# B&R Automation Studio project NewPendant_NG4_11_05_25A (part 16)

```c
					WRST_TML_Param_Set[i].GlbDirection = 1.0;

					WRST_TML_Param_Set[i].MaxAmpl = 0.0;

				break;

			}
		}

		for(i=0 ; i < 1 ; i++){

			switch(i){

				case 0:

					strcpy(Process[PROC_OSC].Name , "OSC");
					strcpy(VectorStateMach[VECT_OSC].Name , "OSC");

					OSC_TML_Param_Set[i].pPrc = &Process[PROC_OSC];
					OSC_TML_Param_Set[i].pVect = &VectorStateMach[VECT_OSC];
					OSC_TML_Param_Set[i].VectStateNum = 1;
					OSC_TML_Param_Set[i].pTML = &TML_MTR_INST[TML_AX_OSC] ;
					OSC_TML_Param_Set[i].Mode = 1; //BPV Mode

					//OSC_TML_Param_Set[i].MaxOscAmpl = 1.0 * 25.4;
					OSC_TML_Param_Set[i].MaxOscAmpl = 0.0;

				break;

			}

		}

		for(i=0 ; i < 1 ; i++){

			switch(i){

				case 0:

					strcpy(Process[PROC_GAS].Name , "GAS");
					GAS_Param_Set[i].pPrc = &Process[PROC_GAS];

					GAS_Param_Set[i].pSensInput     = &Hardware[1].Inp[5];  //FourAxis Head
					GAS_Param_Set[i].pOutput		= &Hardware[1].Outp[4];

				break;

			}

		}

		for(i=0 ; i < 1 ; i++){

			switch(i){

				case 0:

					strcpy(Process[m->pCfg->HeadCfg.INDX.PROC_Indx].Name , "INDX");
					INDEX_Param_Set[i].pPrc = &Process[m->pCfg->HeadCfg.INDX.PROC_Indx];
					//INDEX_Param_Set[i].pPrc = &Process[PROC_INDX];
					INDEX_Param_Set[i].pVect = &VectorStateMach[m->pCfg->HeadCfg.INDX.VECT_A_Indx];
					strcpy(VectorStateMach[m->pCfg->HeadCfg.INDX.VECT_A_Indx].Name , "INDX A");
					strcpy(VectorStateMach[m->pCfg->HeadCfg.INDX.VECT_B_Indx].Name , "INDX B");
					INDEX_Param_Set[i].VectStateNum = 2;
					INDEX_Param_Set[i].Mode = 0;
					INDEX_Param_Set[i].MaxSpeed = 24.0;
					INDEX_Param_Set[i].pCalibPoints		= &m->pCalib->Points[CALIB_TIG_AMPS_CMD];

				break;

			}

		}

		for(i=0 ; i < 1; i++){

			switch(i){

				case 0:

					strcpy(Process[PROC_COOL].Name , "COOLANT");
					COOL_Param_Set[i].pPrc = &Process[PROC_COOL];

					COOL_Param_Set[i].pSensInput     = &Hardware[1].Inp[4];  //FourAxis Head
					COOL_Param_Set[i].pOutput		= &Hardware[1].Outp[6];

				break;

			}

		}

		for(i=0 ; i < 1; i++){

			switch(i){

				case 0:

					strcpy(Process[PROC_HW_PS].Name , "HW PS");
					HW_PS_Param_Set[i].pPrc = &Process[PROC_HW_PS];

					HW_PS_Param_Set[i].pCalibPoints		= &m->pCalib->Points[CALIB_HW_AMPS_CMD];
					HW_PS_Param_Set[i].rawCmdMax 		= 16383.0;
					HW_PS_Param_Set[i].AmpCMD_Max 		= 160.0;

				break;

			}

		}

		for(i=0 ; i < 2; i++){

			switch(i){

				case 0:

					strcpy(Process[PROC_WIRE_FEED].Name ,"WrFeed");
					strcpy(VectorStateMach[VECT_WF].Name ,"WrFeed#1");
					strcpy(VectorStateMach[VECT_WF_1].Name ,"WrFeed#2");

					WIRE_Param_Set[i].pPrc = &Process[PROC_WIRE_FEED];
					WIRE_Param_Set[i].pVect = &VectorStateMach[VECT_WF];
					WIRE_Param_Set[i].VectStateNum = 1; //BPV Mode
					WIRE_Param_Set[i].Mode = 1;
					WIRE_Param_Set[i].MaxSpeedJog = TML_MTR_INST[TML_AX_WF]._cfg.maxVel;

					WIRE_Param_Set[i].pSynchMode = &WFSynchMode;
					WIRE_Param_Set[i].pSynchClock = &SynchClckToWF;

					WIRE_Param_Set[i].pCalibPoints	= &m->pCalib->Points[CALIB_WF_SPEED_CMD];

				break;

				case 1:

					strcpy(Process[PROC_WIRE_PULSE].Name ,"WrPulse");
					strcpy(VectorStateMach[VECT_WP].Name ,"WrPulse#1");
					strcpy(VectorStateMach[VECT_WP_1].Name ,"WrPulse#2");
					WIRE_Param_Set[i].Mode = 1; //BPV Mode

					WIRE_Param_Set[i].pPrc = &Process[PROC_WIRE_PULSE];
					WIRE_Param_Set[i].pVect = &VectorStateMach[VECT_WP];
					WIRE_Param_Set[i].VectStateNum = 1;

					WIRE_Param_Set[i].pSynchMode = &WPSynchMode;
					WIRE_Param_Set[i].pSynchClock = &SynchClckToWP;

					WIRE_Param_Set[i].pCalibPoints	= &m->pCalib->Points[CALIB_WP_SPEED_CMD];

				break;

		}

		}

		for(i=0 ; i < 1; i++){

			switch(i){

				case 0:

					strcpy(Process[PROC_TVL].Name , "TVL");
					strcpy(VectorStateMach[VECT_TVL].Name , "TVL");

					TVL_ROT_Param_Set[i].Mode = 1; //BPV Mode
					TVL_ROT_Param_Set[i].MaxSpeedJog = TML_MTR_INST[TML_AX_TVL]._cfg.maxVel;

					TVL_ROT_Param_Set[i].pPrc = &Process[PROC_TVL];
					TVL_ROT_Param_Set[i].pVect = &VectorStateMach[VECT_TVL];
					TVL_ROT_Param_Set[i].VectStateNum = 1;

					TVL_ROT_Param_Set[i].VectModeForJog = vectSt_Mode_Volt;

					TVL_ROT_Param_Set[i].TotalRescaleFactor = 1.0;
					TVL_ROT_Param_Set[i].pCalibPoints = &m->pCalib->Points[CALIB_TVL_SPEED_CMD];

					TVL_ROT_Param_Set[i].pTrackDia = &curCfg->Param[parTVL_TrackDia].val[0];
					TVL_ROT_Param_Set[i].pVelTolerance = &curCfg->Param[parTVL_SpeedTolerane].val[0];

					// TVL in Torq Mode
					TVL_ROT_Param_Set[i].VectModeForJog = vectSt_Mode_Vel;

					TVL_ROT_Param_Set[i].pEncoder = &AxisCh[TML_AX_TVL].curPos;
					TVL_ROT_Param_Set[i].pHomePos = &OLD_MTR_POS[TVL_ENC_HOME];
					TVL_ROT_Param_Set[i].EncPerTick = m->pCfg->HeadCfg.TVL.EncPerTick;
					TVL_ROT_Param_Set[i].EncDir = m->pCfg->HeadCfg.TVL.Enc_Dir;
					TVL_ROT_Param_Set[i].TicksAtHighVel = 20;

					TVL_ROT_Param_Set[i].pSynchMode = &TVLSynchMode;
					TVL_ROT_Param_Set[i].pSynchClock = &SynchClckToTVL;

			break;

	}

	}

	////////////////////////////////////////////
	/*
	Process[PROC_OSC].Disable = 1;
	Process[PROC_OSC].TestMode = 1;
	VectorStateMach[VECT_OSC].simul = 1;
	TML_MTR_INST[TML_AX_OSC].Disable = 1;
	*/

	Process[PROC_WRST].Disable = 0;
	Process[PROC_WRST].TestMode = 0;
	VectorStateMach[VECT_WRST].simul = 0;
	TML_MTR_INST[TML_AX_WRST].Disable = 0;

	////////////////////////////////////////////////////////////
	/// To jest Tylko do proby
	/*
	VectorStateMach[VECT_AVC].simul = 1;
	VectorStateMach[VECT_OSC].simul = 1;
	VectorStateMach[VECT_TVL].simul = 1;
	VectorStateMach[VECT_INDX_1].simul = 1;
	VectorStateMach[VECT_INDX_2].simul = 1;
	VectorStateMach[VECT_WF_1].simul = 1;
	VectorStateMach[VECT_WF].simul = 1;
	VectorStateMach[VECT_WP_1].simul = 1;
	VectorStateMach[VECT_WP].simul = 1;

	VectorStateMach[VECT_AVC].testMode = 1;
	VectorStateMach[VECT_OSC].testMode = 1;
	VectorStateMach[VECT_TVL].testMode = 1;
	VectorStateMach[VECT_INDX_1].testMode = 1;
	VectorStateMach[VECT_INDX_2].testMode = 1;
	VectorStateMach[VECT_WF_1].testMode = 1;
	VectorStateMach[VECT_WF].testMode = 1;
	VectorStateMach[VECT_WP_1].testMode = 1;
	VectorStateMach[VECT_WP].testMode = 1;

	// To tylko trzeba uncomment gdy jest bez torch ale reszta dziala
	TML_MTR_INST[TML_AX_AVC].Disable = 1;
	TML_MTR_INST[TML_AX_OSC].Disable = 1;
	TML_MTR_INST[TML_AX_TVL].Disable = 1;
	TML_MTR_INST[TML_AX_WRST].Disable = 1;
	TML_MTR_INST[TML_AX_WF].Disable = 1;
	TML_MTR_INST[TML_AX_WF_1].Disable = 1;
	TML_MTR_INST[TML_AX_WP].Disable = 1;
	TML_MTR_INST[TML_AX_WP_1].Disable = 1;
	////////////////////////////////////////

	Process[PROC_AVC].Disable = 1;
	Process[PROC_AVC].TestMode = 1;

	Process[PROC_INDX].Disable = 1;
	Process[PROC_INDX].TestMode = 1;

	Process[PROC_OSC].Disable = 1;
	Process[PROC_OSC].TestMode = 1;

	Process[PROC_TVL].Disable = 1;
	Process[PROC_TVL].TestMode = 1;

	Process[PROC_WIRE_FEED].Disable = 1;
	Process[PROC_WIRE_FEED].TestMode = 1;

	Process[PROC_WIRE_PULSE].Disable = 1;
	Process[PROC_WIRE_PULSE].TestMode = 1;

	Process[PROC_COOL].Disable = 1;
	Process[PROC_COOL].TestMode = 1;

	Process[PROC_GAS].Disable = 1;
	Process[PROC_GAS].TestMode = 1;
	*/
	////////////////////////////////////////////////////////

	return 1;

}

DINT Configure_CLAMSHELL_HEAD(MASTER_typ * m, UINT headType){
int i;

CurCfg_typ *curCfg;
Cfg_typ *cfg;
CurCalib_typ *curCalib , *defaultCalib;

	if(!m)
		return;

	curCfg = (CurCfg_typ*)m->pCurCfg;
	cfg = (Cfg_typ*)m->pCfg;

	curCalib = m->pCalib;
	defaultCalib = m->pDefaultCalib;

	if(!curCfg || !cfg || !curCalib  || !defaultCalib)
		return;

/*********************************************/
	/***   Hardware and Vectors *********************/

	TML_MTR_INST[m->pCfg->HeadCfg.TVL.TML_Indx ].pState = &VectorStateMach[m->pCfg->HeadCfg.TVL.VECT_Indx];

	TML_MTR_INST[m->pCfg->HeadCfg.AVC.TML_A_Indx ].pState = &VectorStateMach[m->pCfg->HeadCfg.AVC.VECT_A_Indx];
	TML_MTR_INST[m->pCfg->HeadCfg.AVC.TML_B_Indx ].pState = &VectorStateMach[m->pCfg->HeadCfg.AVC.VECT_B_Indx];

	TML_MTR_INST[m->pCfg->HeadCfg.OSC.TML_A_Indx ].pState = &VectorStateMach[m->pCfg->HeadCfg.OSC.VECT_A_Indx];
	TML_MTR_INST[m->pCfg->HeadCfg.OSC.TML_B_Indx ].pState = &VectorStateMach[m->pCfg->HeadCfg.OSC.VECT_B_Indx];

	TML_MTR_INST[m->pCfg->HeadCfg.WF.TML_A_Indx ].pState = &VectorStateMach[m->pCfg->HeadCfg.WF.VECT_A_Indx];
	TML_MTR_INST[m->pCfg->HeadCfg.WF.TML_B_Indx ].pState = &VectorStateMach[m->pCfg->HeadCfg.WF.VECT_B_Indx];

	TML_MTR_INST[m->pCfg->HeadCfg.WP.TML_A_Indx ].pState = &VectorStateMach[m->pCfg->HeadCfg.WP.VECT_A_Indx];
	TML_MTR_INST[m->pCfg->HeadCfg.WP.TML_B_Indx ].pState = &VectorStateMach[m->pCfg->HeadCfg.WP.VECT_B_Indx];

	TML_MTR_INST[m->pCfg->HeadCfg.WRST.TML_A_Indx ].pState = &VectorStateMach[m->pCfg->HeadCfg.WRST.VECT_A_Indx];
	TML_MTR_INST[m->pCfg->HeadCfg.WRST.TML_B_Indx ].pState = &VectorStateMach[m->pCfg->HeadCfg.WRST.VECT_B_Indx];

	DC_Mtr[m->pCfg->HeadCfg.INDX.DC_A_Indx ].pState = &VectorStateMach[m->pCfg->HeadCfg.INDX.VECT_A_Indx];
	DC_Mtr[m->pCfg->HeadCfg.INDX.DC_B_Indx ].pState = &VectorStateMach[m->pCfg->HeadCfg.INDX.VECT_B_Indx];

	/*********************************************************/
	/****   Phisical hardware configuration   ************************/

		for(i = 0 ; i < PROCESS_NUM; i++)
			strcpy(Process[i].Name , "spare");

		for(i = 0 ; i < VECTORS_NUM; i++)
			strcpy(VectorStateMach[i].Name , "spare");

			/***********************************/

		//////////////////////////////////////////////////////////////////////////////////
		// Wire Block
		for(i=0 ; i < 2; i++){

			switch(i){

				case 0:
					strcpy(Process[m->pCfg->HeadCfg.WB[i].PROC_Indx].Name , "WB_UD");
					strcpy(VectorStateMach[m->pCfg->HeadCfg.WB[i].VECT_Indx].Name , "WB_UD");

					WR_BLK_Param_Set[i].pPrc = &Process[m->pCfg->HeadCfg.WB[i].PROC_Indx];
					WR_BLK_Param_Set[i].pVect = &VectorStateMach[m->pCfg->HeadCfg.WB[i].VECT_Indx];
					WR_BLK_Param_Set[i].VectStateNum = 1;

					WR_BLK_Param_Set[i].MaxSpeedJog = 24.0;

					Gen_one = 1.0;
					WR_BLK_Param_Set[i].pJogSpeed = &Gen_one;

				break;

				case 1:
					strcpy(Process[m->pCfg->HeadCfg.WB[i].PROC_Indx].Name , "WB_LR");
					strcpy(VectorStateMach[m->pCfg->HeadCfg.WB[i].VECT_Indx].Name , "WB_LR");

					WR_BLK_Param_Set[i].pPrc = &Process[PROC_WB_LR];
					WR_BLK_Param_Set[i].pVect = &VectorStateMach[VECT_WB_LR];
					WR_BLK_Param_Set[i].VectStateNum = 1;

					WR_BLK_Param_Set[i].MaxSpeedJog = 24.0;

					Gen_one = 1.0;
					WR_BLK_Param_Set[i].pJogSpeed = &Gen_one;

				break;

			}

		}

		for(i = 0 ; i < DC2DIRMTR_NUM; i++){

			switch(i){

				case DC_WB_UD:

					strcpy(DC2DirMtr[i].Name , "WB_UD");
					DC2DirMtr[i].pState = &VectorStateMach[VECT_WB_UD];

					DC2DirMtr[i].Cfg.pQ1_output = &Hardware[1].Outp[12];
					DC2DirMtr[i].Cfg.pQ2_output = &Hardware[1].Outp[13];
					DC2DirMtr[i].Cfg.pQ3_output = &Hardware[1].Outp[14];
					DC2DirMtr[i].Cfg.pQ4_output = &Hardware[1].Outp[15];

					DC2DirMtr[i].Cfg.MtrDir = 1.0;

				break;

				case DC_WB_LR:

					strcpy(DC2DirMtr[i].Name , "WB_LR");
					DC2DirMtr[i].pState = &VectorStateMach[VECT_WB_LR];

					DC2DirMtr[i].Cfg.pQ1_output = &Hardware[1].Outp[16];
					DC2DirMtr[i].Cfg.pQ2_output = &Hardware[1].Outp[17];
					DC2DirMtr[i].Cfg.pQ3_output = &Hardware[1].Outp[18];
					DC2DirMtr[i].Cfg.pQ4_output = &Hardware[1].Outp[19];

					DC2DirMtr[i].Cfg.MtrDir = 1.0;

				break;

			}

		}
		/////////////////////////////////////////////////////////////////////////////////

		for(i = 0 ; i < GEN_MTR_NUM; i++){

			switch(i){

				case DC_INDX_1:
				case DC_INDX_2:

					switch(i){

						case DC_INDX_1:

							strcpy(DC_Mtr[i].Name , "DC INDX #1");

							DC_Mtr[i].Cfg.mtr_dir = 1.0;

							if(ProjectConfig == project_US_Orbital) // US Orbital has B and /B swapped
								DC_Mtr[i].Cfg.enc_dir = 1.0;
							else
								DC_Mtr[i].Cfg.enc_dir = -1.0;

							//DC_Mtr[i].Cfg.enc_dir = -1.0;

						break;

						case DC_INDX_2:

							strcpy(DC_Mtr[i].Name , "DC INDX #2");

							DC_Mtr[i].Cfg.mtr_dir = -1.0;

							if(ProjectConfig == project_US_Orbital) // US Orbital has B and /B swapped
								DC_Mtr[i].Cfg.enc_dir = -1.0;
							else
								DC_Mtr[i].Cfg.enc_dir = 1.0;

							//DC_Mtr[i].Cfg.enc_dir = 1.0;

						break;

					}

					//DC_Mtr[i].Cfg.units = 2000 / 59.847340050885561192713356451475; // 2000 enc ticks / 0.75 " dia * 25.4 * PI
					//DC_Mtr[i].Cfg.rev_scale = 66.0 * 0.218686666; // Ratio gear box 66:1

					DC_Mtr[i].Cfg.units =48000 / (1.25 * M_PI * 25.4); // 48000 enc ticks / 1.25 " dia * 25.4 * PI
					DC_Mtr[i].Cfg.rev_scale = 1; // Ratio gear box 66:1

					/* Parameters for PID controller */
					// To nowe
					DC_Mtr[i].msc.PIDParameters.Kp= 100.0;//0.4; //proportional gain / was 0.6
					DC_Mtr[i].msc.PIDParameters.Tn= 0.0;//0.3.1; //intergral action time
					DC_Mtr[i].msc.PIDParameters.Kfbk = 0.1; //windup dampenin

					DC_Mtr[i].msc.PID.enable = 0;
					DC_Mtr[i].msc.PID.pPar = &DC_Mtr[i].msc.PIDParameters;
					DC_Mtr[i].msc.PID.request = 3; // Read parameters from PIDParameters
					DC_Mtr[i].msc.PIDParameters.Tv= 0; //derivative action time
					DC_Mtr[i].msc.PIDParameters.Y_max = 100.0;	//max manipulated variable %
					DC_Mtr[i].msc.PIDParameters.Y_min = -100.0; //min manipulated variable %

				break;

				default:

					strcpy(DC_Mtr[i].Name , "Spare ");

				break;

			}

				//CalcUnits(&DC_Mtr[i]);
				DC_Mtr[i].msc.kPos = (float)DC_Mtr[i].Cfg.units * DC_Mtr[i].Cfg.rev_scale;

		}

		for(i = 0 ; i < TML_SERVO_NUM ; i++){

			switch(i){

				case TML_AX_TVL:

					strcpy(TML_MTR_INST[i].Name , "TVL");

					TML_MTR_INST[i]._cfg.loopPeriod = 0.0005; // Slow loop
					TML_MTR_INST[i]._cfg.units = 1024 * 4; //
					TML_MTR_INST[i]._cfg.rev_motor = 546 * 2; // because loopPeriod is 0.0005
					TML_MTR_INST[i]._cfg.rev_scale = 1.0 /( 2.3 * 25.4 * M_PI) ;

					TML_MTR_INST[i]._cfg.maxVel =  4500.0/60.0/TML_MTR_INST[i]._cfg.rev_motor/ TML_MTR_INST[i]._cfg.rev_scale;
					TML_MTR_INST[i]._cfg.maxAcc = TML_MTR_INST[i]._cfg.maxVel * 10.0 ;
					TML_MTR_INST[i]._cfg.absLastPos = OLD_MTR_POS[TVL_LAST_POS];
					TML_MTR_INST[i]._cfg.absFbk = 2;

					TML_MTR_INST[i]._cfg.HeartBeat = 0.08;

					strcpy(TML_MTR_INST[i]._cfg.programName , "3301_CLMSH_TVL.sw");
					TML_MTR_INST[i].ProgramVersion = ASC2UDINT("3301");

					TML_MTR_INST[i].FirmwareVersion = ASC2UDINT("6A2B");  //0x674B
					TML_MTR_INST[i]._cfg.Appl_ID_adr = 0x7FCF;
					TML_MTR_INST[i]._cfg.NotAutoDownload = 1;

				break;

				case TML_AX_OSC:

					strcpy(TML_MTR_INST[i].Name , "OSC");

					// Analog Feedback from REF
					TML_MTR_INST[i]._cfg.loopPeriod = 0.001;

					TML_MTR_INST[i]._cfg.units = 1024 * 4;
					//TML_MTR_INST[i]._cfg.rev_motor = (-75.0/19.0) * 50.0;
					//TML_MTR_INST[i]._cfg.rev_scale = -1.0/ (0.625 * 25.4 *M_PI) ;
					TML_MTR_INST[i]._cfg.rev_motor = -62;
					TML_MTR_INST[i]._cfg.rev_scale = -1.0/ (0.5 * 25.4) ;

					TML_MTR_INST[i]._cfg.maxVel = 8000.0/60.0/TML_MTR_INST[i]._cfg.rev_motor/ TML_MTR_INST[i]._cfg.rev_scale;
					TML_MTR_INST[i]._cfg.maxAcc = TML_MTR_INST[i]._cfg.maxVel * 10.0 ;
					TML_MTR_INST[i]._cfg.absLastPos = OLD_MTR_POS[OSC_LAST_POS];
					TML_MTR_INST[i]._cfg.absFbk = 2;

					TML_MTR_INST[i]._cfg.HeartBeat = 0.4;
					TML_MTR_INST[i]._cfg.PVTPeriod = 0.08;

					strcpy(TML_MTR_INST[i]._cfg.programName , "3302_CLMSH_OSC.sw");
					TML_MTR_INST[i].ProgramVersion = ASC2UDINT("3302");

					TML_MTR_INST[i].FirmwareVersion = ASC2UDINT("6A2B");
					TML_MTR_INST[i]._cfg.Appl_ID_adr = 0x7FCF;
					TML_MTR_INST[i]._cfg.NotAutoDownload = 1;

					//TML_MTR_INST[i]._cfg.sftLimitPos = curCalib->Points[CALIB_OSC_SFT_LIMIT].val[0];
					//TML_MTR_INST[i]._cfg.sftLimitNeg = curCalib->Points[CALIB_OSC_SFT_LIMIT].val[1];

					//TML_MTR_INST[i]._cfg.sftLimitPos = 0.0;
					//TML_MTR_INST[i]._cfg.sftLimitNeg = 0.0;

				break;

				case TML_AX_AVC:
				case TML_AX_AVC2:

					if(i == TML_AX_AVC)
						strcpy(TML_MTR_INST[i].Name , "AVC");
					else
						strcpy(TML_MTR_INST[i].Name , "AVC_2");

					// Analog Feedback from REF
					TML_MTR_INST[i]._cfg.loopPeriod = 0.001;
					TML_MTR_INST[i]._cfg.units = 4096;
					TML_MTR_INST[i]._cfg.rev_motor = 1;
					TML_MTR_INST[i]._cfg.rev_scale = 1.0/5.0;
					TML_MTR_INST[i]._cfg.maxVel = 1500.0;
					TML_MTR_INST[i]._cfg.maxAcc = TML_MTR_INST[i]._cfg.maxVel * 10.0;
					//TML_MTR_INST[i]._cfg.satpMax = 27853; // KPP bylo Stauration of proportional gain
					TML_MTR_INST[i]._cfg.satpMax = 32000; // KPP bylo Stauration of proportional gain
					//TML_MTR_INST[i]._cfg.kppMax = 32000; // KPP bylo Stauration of proportional gain
					//TML_MTR_INST[i]._cfg.kipMax = 200; // KPP bylo Stauration of proportional gain
					TML_MTR_INST[i]._cfg.kppMax = 32000;
					TML_MTR_INST[i]._cfg.kipMax = 1000;
					TML_MTR_INST[i]._cfg.absFbk = 0;

					TML_MTR_INST[i]._cfg.HeartBeat = 0.8;

					TML_MTR_INST[i]._cfg.signFilter = curCfg->Param[parAVC_FbkFilter].val[0];

					//U_BEND_HP_PINS
					strcpy(TML_MTR_INST[i]._cfg.programName , "3303_CLMSH_AVC.sw");
					TML_MTR_INST[i].ProgramVersion = ASC2UDINT("3303");

					TML_MTR_INST[i].FirmwareVersion = ASC2UDINT("6A2B");  //0x674C , 514D
					TML_MTR_INST[i]._cfg.Appl_ID_adr = 0x7FCF;
					TML_MTR_INST[i]._cfg.NotAutoDownload = 1;

					//TML_MTR_INST[i]._cfg.sftLimitPos = 0.0;
					//TML_MTR_INST[i]._cfg.sftLimitNeg = 0.0;

					/*
					TML_MTR_INST[i]._cfg.AnalLimitPos = 3900;
					TML_MTR_INST[i]._cfg.AnalLimitNeg = 100;
					*/

					TML_MTR_INST[i]._cfg.AnalLimitPos = 0;
					TML_MTR_INST[i]._cfg.AnalLimitNeg = 0;

				break;

				// WRIST
				case TML_AX_WF_1: //TML_AX_WRST:

					strcpy(TML_MTR_INST[i].Name , "WRIST");

					// Analog Feedback from REF
					TML_MTR_INST[i]._cfg.loopPeriod = 0.001;

					TML_MTR_INST[i]._cfg.units = 1024 * 4;
					//TML_MTR_INST[i]._cfg.rev_motor = (-75.0/19.0) * 50.0;
					//TML_MTR_INST[i]._cfg.rev_scale = -1.0/ (0.625 * 25.4 *M_PI) ;
					TML_MTR_INST[i]._cfg.rev_motor = 16 * 50;
					TML_MTR_INST[i]._cfg.rev_scale = 1.0/ (360.0) ;

					TML_MTR_INST[i]._cfg.maxVel = 8000.0/60.0/TML_MTR_INST[i]._cfg.rev_motor/ TML_MTR_INST[i]._cfg.rev_scale;
					TML_MTR_INST[i]._cfg.maxAcc = TML_MTR_INST[i]._cfg.maxVel * 10.0 ;
					TML_MTR_INST[i]._cfg.absLastPos = OLD_MTR_POS[WRST_LAST_POS];
					TML_MTR_INST[i]._cfg.absFbk = 0;
					//TML_MTR_INST[i]._cfg.absFbk = 2;

					TML_MTR_INST[i]._cfg.HeartBeat = 0.02;
					TML_MTR_INST[i]._cfg.PVTPeriod = 0.08;

					strcpy(TML_MTR_INST[i]._cfg.programName , "3307_CLMSH_WRST.sw");
					TML_MTR_INST[i].ProgramVersion = ASC2UDINT("3307");

					TML_MTR_INST[i].FirmwareVersion = ASC2UDINT("6A2B");
					TML_MTR_INST[i]._cfg.Appl_ID_adr = 0x7FCF;
					TML_MTR_INST[i]._cfg.NotAutoDownload = 1;

					//TML_MTR_INST[i]._cfg.sftLimitPos = curCalib->Points[CALIB_OSC_SFT_LIMIT].val[0];
					//TML_MTR_INST[i]._cfg.sftLimitNeg = curCalib->Points[CALIB_OSC_SFT_LIMIT].val[1];

					//TML_MTR_INST[i]._cfg.sftLimitPos = 0.0;
					//TML_MTR_INST[i]._cfg.sftLimitNeg = 0.0;

				break;

				case TML_AX_WF:

					strcpy(TML_MTR_INST[i].Name , "WF");
					TML_MTR_INST[i]._cfg.rev_scale = 1.0 /( 0.75 * 25.4 * M_PI) ;
					TML_MTR_INST[i]._cfg.rev_motor = 35.0;	// jest 39:1 ale trzeba pamietac o groove na rolce

					// Analog Feedback from REF
					TML_MTR_INST[i]._cfg.loopPeriod = 0.001;
					TML_MTR_INST[i]._cfg.units = 1024 * 4; //
					//TML_MTR_INST[i]._cfg.rev_motor = 35;

					TML_MTR_INST[i]._cfg.maxVel = 520 * 25.4/ 60.0; //// 520 ipm
					//TML_MTR_INST[i]._cfg.maxAcc = TML_MTR_INST[i]._cfg.maxVel * 100.0;
					TML_MTR_INST[i]._cfg.maxAcc = TML_MTR_INST[i]._cfg.maxVel * 4.0;
					TML_MTR_INST[i]._cfg.absFbk = 0;

					TML_MTR_INST[i]._cfg.HeartBeat = 0.4;

					strcpy(TML_MTR_INST[i]._cfg.programName , "3305_CLMSH_WF.sw");
					TML_MTR_INST[i].ProgramVersion = ASC2UDINT("3305");

					TML_MTR_INST[i].FirmwareVersion = ASC2UDINT("6A2B");
					TML_MTR_INST[i]._cfg.Appl_ID_adr = 0x7FCF;
					TML_MTR_INST[i]._cfg.NotAutoDownload = 1;

				break;

				case TML_AX_WP:

					strcpy(TML_MTR_INST[i].Name , "WP");

					// Analog Feedback from REF
					TML_MTR_INST[i]._cfg.loopPeriod = 0.001;

					TML_MTR_INST[i]._cfg.units = 1024 * 4;
					TML_MTR_INST[i]._cfg.rev_motor = 3.9;
					TML_MTR_INST[i]._cfg.rev_scale = 1.0/2.0;

					/*
					TML_MTR_INST[i]._cfg.units = 500 * 4;
					TML_MTR_INST[i]._cfg.rev_motor = 24;
					TML_MTR_INST[i]._cfg.rev_scale = 1.0/5.0;
					*/

					TML_MTR_INST[i]._cfg.maxVel = 10000.0; //
					TML_MTR_INST[i]._cfg.maxAcc = 100.0;
					TML_MTR_INST[i]._cfg.absFbk = 0;

					TML_MTR_INST[i]._cfg.HeartBeat = 0.4;

					strcpy(TML_MTR_INST[i]._cfg.programName , "3306_CLMSH_WP.sw");
					TML_MTR_INST[i].ProgramVersion = ASC2UDINT("3306");

					TML_MTR_INST[i].FirmwareVersion = ASC2UDINT("6A2B");
					TML_MTR_INST[i]._cfg.Appl_ID_adr = 0x7FCF;
					TML_MTR_INST[i]._cfg.NotAutoDownload = 1;

				break;

				default:

					//strcpy(TML_MTR_INST[i].Name , "Spare ");
					xsprintf(TML_MTR_INST[i].Name, "Spare %d", i );

				break;

			}

		TML_MTR_INST[i].xCMD = TML_RESTART;

	}

		TML_mgr[0].hrdw[0].AxisNum = 0;
		TML_mgr[0].hrdw[1].AxisNum = 7;

		TML_mgr[0].pAxis[0] = &AxisCh[TML_mgr[0].hrdw[0].AxisNum];
		TML_mgr[0].pAxis[1] = &AxisCh[TML_mgr[0].hrdw[0].AxisNum];
		//TML_mgr[0].pAxis[1] = &AxisCh[TML_mgr[0].hrdw[1].AxisNum];

		TML_mgr[0].pTML[0] = &TML_MTR_INST[0];
		TML_mgr[0].pTML[1] = &TML_MTR_INST[TML_mgr[0].hrdw[0].AxisNum];

		AxisCh[TML_AX_TVL].AxisID	= 1;
		AxisCh[TML_AX_OSC].AxisID 	= 2;
		AxisCh[TML_AX_AVC].AxisID 	= 3;
		AxisCh[TML_AX_AVC2].AxisID 	= 4;

		AxisCh[TML_AX_WF].AxisID 	= 5;
		AxisCh[TML_AX_WP].AxisID 	= 6;

		AxisCh[m->pCfg->HeadCfg.WRST.TML_A_Indx].AxisID 	= 7;

		//AxisCh[TML_AX_WF_1].AxisID 	= 7;
		//AxisCh[TML_AX_WP_1].AxisID 	= 8;
		/**************************************/
		/****   Process   ************************/

		// Lincoln Power Supply
		for(i=0 ; i < 1; i++){

			switch(i){

				case 0:

					strcpy(Process[PROC_TIG_PS].Name , "TIG PS");
					PS_Param_Set[i].pPrc = &Process[PROC_TIG_PS];

					PS_Param_Set[i].pCalibPoints		= &m->pCalib->Points[CALIB_TIG_AMPS_CMD];
					//PS_Param_Set[i].rawCmdMax			= 26170; // //
					//PS_Param_Set[i].AmpCMD_Max			= 500.0; // 62.5 amp / 1 V
					PS_Param_Set[i].rawCmdMax			= 32767;
					PS_Param_Set[i].AmpCMD_Max			= 627.0;

					PS_Param_Set[i].pArcLinkRobot   = (UDINT)&ArcLink.robot;

					PS_Param_Set[i].Mode 			= 1; // Arclink connection

				break;

			}

		}
		///////////////////////////////////////////////////////

		for(i=0 ; i < 1 ; i++){

			switch(i){

				case 0:

					strcpy(Process[PROC_AVC].Name , "AVC");

					strcpy(VectorStateMach[VECT_AVC].Name , "AVC");
					strcpy(VectorStateMach[VECT_AVC2].Name , "AVC_2");

					AVC_Param_Set[i].pPrc = &Process[PROC_AVC];
					AVC_Param_Set[i].pVect = &VectorStateMach[VECT_AVC];
					AVC_Param_Set[i].VectStateNum = 2;
					AVC_Param_Set[i].Mode = 1; //BPV Mode
					AVC_Param_Set[i].Mode = 3; //BPV Mode w/ twp torches
					AVC_Param_Set[i].MaxSpeedJog = TML_MTR_INST[TML_AX_AVC]._cfg.maxVel;

					m->pCalib->Points[CALIB_TIG_VOLT_FBK].num = 10;
					AVC_Param_Set[i].pCalibPoints		= &m->pCalib->Points[CALIB_TIG_VOLT_FBK];

				break;

			}
		}

		for(i=0 ; i < 1 ; i++){

			switch(i){

				case 0:

					strcpy(Process[m->pCfg->HeadCfg.WRST.PROC_Indx].Name , "WRST");
					strcpy(VectorStateMach[m->pCfg->HeadCfg.WRST.VECT_A_Indx].Name , "WRST");

					WRST_TML_Param_Set[i].pPrc = &Process[m->pCfg->HeadCfg.WRST.PROC_Indx];
					WRST_TML_Param_Set[i].pVect = &VectorStateMach[m->pCfg->HeadCfg.WRST.VECT_A_Indx];
					WRST_TML_Param_Set[i].VectStateNum = 1;
					WRST_TML_Param_Set[i].pTML = &TML_MTR_INST[m->pCfg->HeadCfg.WRST.TML_A_Indx] ;
					WRST_TML_Param_Set[i].Mode = 10; // ClamShell Head  mode with Wrist

					WRST_TML_Param_Set[i].GlbDirection = 1.0;

					WRST_TML_Param_Set[i].MaxAmpl = 0.0;

				break;

			}
		}

		for(i=0 ; i < 1 ; i++){

			switch(i){

				case 0:

					strcpy(Process[PROC_OSC].Name , "OSC");
					strcpy(VectorStateMach[VECT_OSC].Name , "OSC");

					OSC_TML_Param_Set[i].pPrc = &Process[PROC_OSC];
					OSC_TML_Param_Set[i].pVect = &VectorStateMach[VECT_OSC];
					OSC_TML_Param_Set[i].VectStateNum = 1;
					OSC_TML_Param_Set[i].pTML = &TML_MTR_INST[TML_AX_OSC] ;
					OSC_TML_Param_Set[i].Mode = 1; //BPV Mode

					//OSC_TML_Param_Set[i].MaxOscAmpl = 1.0 * 25.4;
					OSC_TML_Param_Set[i].MaxOscAmpl = 0.0;

				break;

			}

		}

		for(i=0 ; i < 1 ; i++){

			switch(i){

				case 0:

					strcpy(Process[PROC_GAS].Name , "GAS");
					GAS_Param_Set[i].pPrc = &Process[PROC_GAS];

					//GAS_Param_Set[i].pSensInput     = &Hardware[1].Inp[5];  //FourAxis Head
					//GAS_Param_Set[i].pOutput		= &Hardware[1].Outp[4];

					GAS_Param_Set[i].Mode = 1;// Arclik Gas Sol

				break;

			}

		}

		for(i=0 ; i < 1 ; i++){

			switch(i){

				case 0:

					strcpy(Process[m->pCfg->HeadCfg.INDX.PROC_Indx].Name , "INDX");
					INDEX_Param_Set[i].pPrc = &Process[m->pCfg->HeadCfg.INDX.PROC_Indx];
					//INDEX_Param_Set[i].pPrc = &Process[PROC_INDX];
					INDEX_Param_Set[i].pVect = &VectorStateMach[m->pCfg->HeadCfg.INDX.VECT_A_Indx];
					strcpy(VectorStateMach[m->pCfg->HeadCfg.INDX.VECT_A_Indx].Name , "INDX A");
					strcpy(VectorStateMach[m->pCfg->HeadCfg.INDX.VECT_B_Indx].Name , "INDX B");
					INDEX_Param_Set[i].VectStateNum = 2;
					INDEX_Param_Set[i].Mode = 0;
					INDEX_Param_Set[i].MaxSpeed = 24.0;
					INDEX_Param_Set[i].pCalibPoints		= &m->pCalib->Points[CALIB_TIG_AMPS_CMD];

				break;

			}

		}

		for(i=0 ; i < 1; i++){

			switch(i){

				case 0:

					strcpy(Process[PROC_COOL].Name , "COOLANT");
					COOL_Param_Set[i].pPrc = &Process[PROC_COOL];

					//COOL_Param_Set[i].pSensInput     = &Hardware[1].Inp[4];  //FourAxis Head
					//COOL_Param_Set[i].pOutput		= &Hardware[1].Outp[6];

				break;

			}

		}

		for(i=0 ; i < 1; i++){

			switch(i){

				case 0:

					strcpy(Process[PROC_HW_PS].Name , "HW PS");
					HW_PS_Param_Set[i].pPrc = &Process[PROC_HW_PS];

					HW_PS_Param_Set[i].pCalibPoints		= &m->pCalib->Points[CALIB_HW_AMPS_CMD];

					// small Jack PS
					HW_PS_Param_Set[i].rawCmdMax 		= 16383.0;
					HW_PS_Param_Set[i].AmpCMD_Max 		= 160.0;

					// Lincoln PS
					//HW_PS_Param_Set[i].rawCmdMax 		= 32767.0;
					//HW_PS_Param_Set[i].AmpCMD_Max 		= 160.0;

					HW_PS_Param_Set[i].pAnal_Output 	= &Hardware[1].Anal_Outp[0]; // HotwirePS_AO
					HW_PS_Param_Set[i].pOutput			= &Hardware[1].Outp[2]; //HotwirePS_Enable

				break;

			}

		}

		for(i=0 ; i < 2; i++){

			switch(i){

				case 0:

					strcpy(Process[PROC_WIRE_FEED].Name ,"WrFeed");
					strcpy(VectorStateMach[VECT_WF].Name ,"WrFeed#1");
					strcpy(VectorStateMach[VECT_WF_1].Name ,"WrFeed#2");

					WIRE_Param_Set[i].pPrc = &Process[PROC_WIRE_FEED];
					WIRE_Param_Set[i].pVect = &VectorStateMach[VECT_WF];
					WIRE_Param_Set[i].VectStateNum = 1;
					WIRE_Param_Set[i].Mode = 3; //BPV Mode with Feedback Selection
					WIRE_Param_Set[i].MaxSpeedJog = TML_MTR_INST[TML_AX_WF]._cfg.maxVel;

					WIRE_Param_Set[i].pSynchMode = &WFSynchMode;
					WIRE_Param_Set[i].pSynchClock = &SynchClckToWF;

					WIRE_Param_Set[i].pCalibPoints	= &m->pCalib->Points[CALIB_WF_SPEED_CMD];

				break;

				case 1:

					strcpy(Process[PROC_WIRE_PULSE].Name ,"WrPulse");
					strcpy(VectorStateMach[VECT_WP].Name ,"WrPulse#1");
					strcpy(VectorStateMach[VECT_WP_1].Name ,"WrPulse#2");
					WIRE_Param_Set[i].Mode = 3; //BPV Mode with Feedback Selection

					WIRE_Param_Set[i].pPrc = &Process[PROC_WIRE_PULSE];
					WIRE_Param_Set[i].pVect = &VectorStateMach[VECT_WP];
					WIRE_Param_Set[i].VectStateNum = 1;

					WIRE_Param_Set[i].pSynchMode = &WPSynchMode;
					WIRE_Param_Set[i].pSynchClock = &SynchClckToWP;

					WIRE_Param_Set[i].pCalibPoints	= &m->pCalib->Points[CALIB_WP_SPEED_CMD];

				break;

		}

	}

		for(i=0 ; i < 1; i++){

			switch(i){

				case 0:

					strcpy(Process[PROC_TVL].Name , "TVL");
					strcpy(VectorStateMach[VECT_TVL].Name , "TVL");

					//TVL_ROT_Param_Set[i].Mode = 1; //BPV Mode
					TVL_ROT_Param_Set[i].Mode = 2;  //TVL_MODE_BPV_PosMode
					TVL_ROT_Param_Set[i].MaxSpeedJog = TML_MTR_INST[TML_AX_TVL]._cfg.maxVel;

					TVL_ROT_Param_Set[i].pPrc = &Process[PROC_TVL];
					TVL_ROT_Param_Set[i].pVect = &VectorStateMach[VECT_TVL];
					TVL_ROT_Param_Set[i].VectStateNum = 1;

					TVL_ROT_Param_Set[i].VectModeForJog = vectSt_Mode_Volt;

					TVL_ROT_Param_Set[i].TotalRescaleFactor = 1.0;
					TVL_ROT_Param_Set[i].pCalibPoints = &m->pCalib->Points[CALIB_TVL_SPEED_CMD];

					TVL_ROT_Param_Set[i].pTrackDia = &curCfg->Param[parTVL_TrackDia].val[0];
					TVL_ROT_Param_Set[i].pVelTolerance = &curCfg->Param[parTVL_SpeedTolerane].val[0];

					// TVL in Torq Mode
					TVL_ROT_Param_Set[i].VectModeForJog = vectSt_Mode_Vel;

					TVL_ROT_Param_Set[i].pEncoder = &AxisCh[TML_AX_TVL].curPos;
					TVL_ROT_Param_Set[i].pHomePos = &OLD_MTR_POS[TVL_ENC_HOME];
					TVL_ROT_Param_Set[i].EncPerTick = m->pCfg->HeadCfg.TVL.EncPerTick;
					TVL_ROT_Param_Set[i].EncDir = m->pCfg->HeadCfg.TVL.Enc_Dir;
					TVL_ROT_Param_Set[i].TicksAtHighVel = 20;

					TVL_ROT_Param_Set[i].pSynchMode = &TVLSynchMode;
					TVL_ROT_Param_Set[i].pSynchClock = &SynchClckToTVL;

			break;

	}

	}

	////////////////////////////////////////////

	////////////////////////////////////////////////////////////
	/// To jest Tylko do proby

	/*
	VectorStateMach[VECT_AVC].simul = 1;
	VectorStateMach[VECT_AVC2].simul = 1;
	VectorStateMach[VECT_OSC].simul = 1;
	VectorStateMach[VECT_TVL].simul = 1;
	VectorStateMach[VECT_INDX_1].simul = 1;
	VectorStateMach[VECT_INDX_2].simul = 1;
	VectorStateMach[VECT_WF_1].simul = 1;
	VectorStateMach[VECT_WF].simul = 1;
	VectorStateMach[VECT_WP_1].simul = 1;
	VectorStateMach[VECT_WP].simul = 1;
	VectorStateMach[VECT_WRST].simul = 1;

	VectorStateMach[VECT_AVC].testMode = 1;
	VectorStateMach[VECT_AVC2].testMode = 1;
	VectorStateMach[VECT_OSC].testMode = 1;
	VectorStateMach[VECT_TVL].testMode = 1;
	VectorStateMach[VECT_INDX_1].testMode = 1;
	VectorStateMach[VECT_INDX_2].testMode = 1;
	VectorStateMach[VECT_WF_1].testMode = 1;
	VectorStateMach[VECT_WF].testMode = 1;
	VectorStateMach[VECT_WP_1].testMode = 1;
	VectorStateMach[VECT_WP].testMode = 1;
	VectorStateMach[VECT_WRST].testMode = 1;
	*/

	// To tylko trzeba uncomment gdy jest bez torch ale reszta dziala

	//TML_MTR_INST[TML_AX_AVC].Disable = 1;
	//TML_MTR_INST[TML_AX_AVC2].Disable = 1;
	//TML_MTR_INST[TML_AX_OSC].Disable = 1;
	//TML_MTR_INST[TML_AX_TVL].Disable = 1;
	//TML_MTR_INST[TML_AX_WRST].Disable = 1;
	//TML_MTR_INST[TML_AX_WF].Disable = 1;
	//TML_MTR_INST[TML_AX_WF_1].Disable = 1;
	//TML_MTR_INST[TML_AX_WP].Disable = 1;
	//TML_MTR_INST[TML_AX_WP_1].Disable = 1;

	////////////////////////////////////////

	//Process[PROC_AVC].Disable = 1;
	//Process[PROC_AVC].TestMode = 1;

	//Process[PROC_INDX].Disable = 1;
	//Process[PROC_INDX].TestMode = 1;

	//Process[PROC_OSC].Disable = 1;
	//Process[PROC_OSC].TestMode = 1;

	//Process[PROC_WRST].Disable = 1;
	//Process[PROC_WRST].TestMode = 1;

	//Process[PROC_TVL].Disable = 1;
	//Process[PROC_TVL].TestMode = 1;

	//Process[PROC_WIRE_FEED].Disable = 1;
	//Process[PROC_WIRE_FEED].TestMode = 1;

	//Process[PROC_WIRE_PULSE].Disable = 1;
	//Process[PROC_WIRE_PULSE].TestMode = 1;

	//Process[PROC_COOL].Disable = 1;
	//Process[PROC_COOL].TestMode = 1;

	//Process[PROC_GAS].Disable = 1;
	//Process[PROC_GAS].TestMode = 1;

	////////////////////////////////////////////////////////

	return 1;

}

DINT Configure_CHERRYPOINT_BPV1_HEAD(MASTER_typ * m, UINT headType){
int i;

CurCfg_typ *curCfg;
Cfg_typ *cfg;
CurCalib_typ *curCalib , *defaultCalib;

	if(!m)
		return;

	curCfg = (CurCfg_typ*)m->pCurCfg;
	cfg = (Cfg_typ*)m->pCfg;

	curCalib = m->pCalib;
	defaultCalib = m->pDefaultCalib;

	if(!curCfg || !cfg || !curCalib  || !defaultCalib)
		return;

/*********************************************/
	/***   Hardware and Vectors *********************/

	TML_MTR_INST[m->pCfg->HeadCfg.TVL.TML_Indx ].pState = &VectorStateMach[m->pCfg->HeadCfg.TVL.VECT_Indx];

	TML_MTR_INST[m->pCfg->HeadCfg.AVC.TML_A_Indx ].pState = &VectorStateMach[m->pCfg->HeadCfg.AVC.VECT_A_Indx];
	TML_MTR_INST[m->pCfg->HeadCfg.AVC.TML_B_Indx ].pState = &VectorStateMach[m->pCfg->HeadCfg.AVC.VECT_B_Indx];

	TML_MTR_INST[m->pCfg->HeadCfg.OSC.TML_A_Indx ].pState = &VectorStateMach[m->pCfg->HeadCfg.OSC.VECT_A_Indx];
	TML_MTR_INST[m->pCfg->HeadCfg.OSC.TML_B_Indx ].pState = &VectorStateMach[m->pCfg->HeadCfg.OSC.VECT_B_Indx];

	TML_MTR_INST[m->pCfg->HeadCfg.WF.TML_A_Indx ].pState = &VectorStateMach[m->pCfg->HeadCfg.WF.VECT_A_Indx];
	TML_MTR_INST[m->pCfg->HeadCfg.WF.TML_B_Indx ].pState = &VectorStateMach[m->pCfg->HeadCfg.WF.VECT_B_Indx];

	TML_MTR_INST[m->pCfg->HeadCfg.WP.TML_A_Indx ].pState = &VectorStateMach[m->pCfg->HeadCfg.WP.VECT_A_Indx];
	TML_MTR_INST[m->pCfg->HeadCfg.WP.TML_B_Indx ].pState = &VectorStateMach[m->pCfg->HeadCfg.WP.VECT_B_Indx];

	TML_MTR_INST[m->pCfg->HeadCfg.WRST.TML_A_Indx ].pState = &VectorStateMach[m->pCfg->HeadCfg.WRST.VECT_A_Indx];
	TML_MTR_INST[m->pCfg->HeadCfg.WRST.TML_B_Indx ].pState = &VectorStateMach[m->pCfg->HeadCfg.WRST.VECT_B_Indx];

	DC_Mtr[m->pCfg->HeadCfg.INDX.DC_A_Indx ].pState = &VectorStateMach[m->pCfg->HeadCfg.INDX.VECT_A_Indx];
	DC_Mtr[m->pCfg->HeadCfg.INDX.DC_B_Indx ].pState = &VectorStateMach[m->pCfg->HeadCfg.INDX.VECT_B_Indx];

	/*********************************************************/
	/****   Phisical hardware configuration   ************************/

		for(i = 0 ; i < PROCESS_NUM; i++)
			strcpy(Process[i].Name , "spare");

		for(i = 0 ; i < VECTORS_NUM; i++)
			strcpy(VectorStateMach[i].Name , "spare");

			/***********************************/

		//////////////////////////////////////////////////////////////////////////////////
		// Wire Block
		for(i=0 ; i < 2; i++){

			switch(i){

				case 0:
					strcpy(Process[m->pCfg->HeadCfg.WB[i].PROC_Indx].Name , "WB_UD");
					strcpy(VectorStateMach[m->pCfg->HeadCfg.WB[i].VECT_Indx].Name , "WB_UD");

					WR_BLK_Param_Set[i].pPrc = &Process[m->pCfg->HeadCfg.WB[i].PROC_Indx];
					WR_BLK_Param_Set[i].pVect = &VectorStateMach[m->pCfg->HeadCfg.WB[i].VECT_Indx];
					WR_BLK_Param_Set[i].VectStateNum = 1;

					WR_BLK_Param_Set[i].MaxSpeedJog = 24.0;

					Gen_one = 1.0;
					WR_BLK_Param_Set[i].pJogSpeed = &Gen_one;

				break;

				case 1:
					strcpy(Process[m->pCfg->HeadCfg.WB[i].PROC_Indx].Name , "WB_LR");
					strcpy(VectorStateMach[m->pCfg->HeadCfg.WB[i].VECT_Indx].Name , "WB_LR");

					WR_BLK_Param_Set[i].pPrc = &Process[PROC_WB_LR];
					WR_BLK_Param_Set[i].pVect = &VectorStateMach[VECT_WB_LR];
					WR_BLK_Param_Set[i].VectStateNum = 1;

					WR_BLK_Param_Set[i].MaxSpeedJog = 24.0;

					Gen_one = 1.0;
					WR_BLK_Param_Set[i].pJogSpeed = &Gen_one;

				break;

			}

		}

		for(i = 0 ; i < DC2DIRMTR_NUM; i++){

			switch(i){

				case DC_WB_UD:

					strcpy(DC2DirMtr[i].Name , "WB_UD");
					DC2DirMtr[i].pState = &VectorStateMach[VECT_WB_UD];

					DC2DirMtr[i].Cfg.pQ1_output = &Hardware[1].Outp[12];
					DC2DirMtr[i].Cfg.pQ2_output = &Hardware[1].Outp[13];
					DC2DirMtr[i].Cfg.pQ3_output = &Hardware[1].Outp[14];
					DC2DirMtr[i].Cfg.pQ4_output = &Hardware[1].Outp[15];

					DC2DirMtr[i].Cfg.MtrDir = 1.0;

				break;

				case DC_WB_LR:

					strcpy(DC2DirMtr[i].Name , "WB_LR");
					DC2DirMtr[i].pState = &VectorStateMach[VECT_WB_LR];

					DC2DirMtr[i].Cfg.pQ1_output = &Hardware[1].Outp[16];
					DC2DirMtr[i].Cfg.pQ2_output = &Hardware[1].Outp[17];
					DC2DirMtr[i].Cfg.pQ3_output = &Hardware[1].Outp[18];
					DC2DirMtr[i].Cfg.pQ4_output = &Hardware[1].Outp[19];

					DC2DirMtr[i].Cfg.MtrDir = 1.0;

				break;

			}

		}
		/////////////////////////////////////////////////////////////////////////////////

		for(i = 0 ; i < GEN_MTR_NUM; i++){

			switch(i){

				case DC_INDX_1:
				case DC_INDX_2:

					switch(i){

						case DC_INDX_1:

							strcpy(DC_Mtr[i].Name , "DC INDX #1");

							DC_Mtr[i].Cfg.mtr_dir = 1.0;

							if(ProjectConfig == project_US_Orbital) // US Orbital has B and /B swapped
								DC_Mtr[i].Cfg.enc_dir = 1.0;
							else
								DC_Mtr[i].Cfg.enc_dir = -1.0;

							//DC_Mtr[i].Cfg.enc_dir = -1.0;

						break;

						case DC_INDX_2:

							strcpy(DC_Mtr[i].Name , "DC INDX #2");

							DC_Mtr[i].Cfg.mtr_dir = -1.0;

							if(ProjectConfig == project_US_Orbital) // US Orbital has B and /B swapped
								DC_Mtr[i].Cfg.enc_dir = -1.0;
							else
								DC_Mtr[i].Cfg.enc_dir = 1.0;

							//DC_Mtr[i].Cfg.enc_dir = 1.0;

						break;

					}

					//DC_Mtr[i].Cfg.units = 2000 / 59.847340050885561192713356451475; // 2000 enc ticks / 0.75 " dia * 25.4 * PI
					//DC_Mtr[i].Cfg.rev_scale = 66.0 * 0.218686666; // Ratio gear box 66:1

					DC_Mtr[i].Cfg.units =48000 / (1.25 * M_PI * 25.4); // 48000 enc ticks / 1.25 " dia * 25.4 * PI
					DC_Mtr[i].Cfg.rev_scale = 1; // Ratio gear box 66:1

					/* Parameters for PID controller */
					// To nowe
					DC_Mtr[i].msc.PIDParameters.Kp= 100.0;//0.4; //proportional gain / was 0.6
					DC_Mtr[i].msc.PIDParameters.Tn= 0.0;//0.3.1; //intergral action time
					DC_Mtr[i].msc.PIDParameters.Kfbk = 0.1; //windup dampenin

					DC_Mtr[i].msc.PID.enable = 0;
					DC_Mtr[i].msc.PID.pPar = &DC_Mtr[i].msc.PIDParameters;
					DC_Mtr[i].msc.PID.request = 3; // Read parameters from PIDParameters
					DC_Mtr[i].msc.PIDParameters.Tv= 0; //derivative action time
					DC_Mtr[i].msc.PIDParameters.Y_max = 100.0;	//max manipulated variable %
					DC_Mtr[i].msc.PIDParameters.Y_min = -100.0; //min manipulated variable %

				break;

				default:

					strcpy(DC_Mtr[i].Name , "Spare ");

				break;

			}

				//CalcUnits(&DC_Mtr[i]);
				DC_Mtr[i].msc.kPos = (float)DC_Mtr[i].Cfg.units * DC_Mtr[i].Cfg.rev_scale;

		}

		for(i = 0 ; i < TML_SERVO_NUM ; i++){

			switch(i){

				case TML_AX_TVL:

					strcpy(TML_MTR_INST[i].Name , "TVL");

					TML_MTR_INST[i]._cfg.loopPeriod = 0.0005; // Slow loop
					TML_MTR_INST[i]._cfg.units = 1024 * 4; //
					TML_MTR_INST[i]._cfg.rev_motor = 156;
					TML_MTR_INST[i]._cfg.rev_scale = 1.0 /( 1.25 * 25.4 * M_PI) ;

					TML_MTR_INST[i]._cfg.maxVel =  fabsf(4500.0/60.0/TML_MTR_INST[i]._cfg.rev_motor/ TML_MTR_INST[i]._cfg.rev_scale);
					TML_MTR_INST[i]._cfg.maxAcc = TML_MTR_INST[i]._cfg.maxVel * 10.0 ;
					TML_MTR_INST[i]._cfg.absLastPos = OLD_MTR_POS[TVL_LAST_POS];
					TML_MTR_INST[i]._cfg.absFbk = 2;

					TML_MTR_INST[i]._cfg.HeartBeat = 0.08;

					strcpy(TML_MTR_INST[i]._cfg.programName , "0331_BPV_TVL.sw");
					TML_MTR_INST[i].ProgramVersion = ASC2UDINT("0331");

					TML_MTR_INST[i].FirmwareVersion = ASC2UDINT("6A2B");  //0x674B
					TML_MTR_INST[i]._cfg.Appl_ID_adr = 0x7FCF;
					TML_MTR_INST[i]._cfg.NotAutoDownload = 1;

				break;

				case TML_AX_OSC:

					strcpy(TML_MTR_INST[i].Name , "OSC");

					TML_MTR_INST[i]._cfg.loopPeriod = 0.001;

					TML_MTR_INST[i]._cfg.units = 1024 * 4;

					TML_MTR_INST[i]._cfg.rev_motor = -75.0/19.0;
					//TML_MTR_INST[i]._cfg.rev_scale = -1.0/ (0.625 * 25.4 *M_PI) ;
					TML_MTR_INST[i]._cfg.rev_scale = 1.0/ ((1.0/8.0) * 25.4) ;

					TML_MTR_INST[i]._cfg.maxVel = 8000.0/60.0/TML_MTR_INST[i]._cfg.rev_motor/ TML_MTR_INST[i]._cfg.rev_scale;

					TML_MTR_INST[i]._cfg.absLastPos = OLD_MTR_POS[OSC_LAST_POS];
					TML_MTR_INST[i]._cfg.pAbsLastPos = &OLD_MTR_POS[OSC_LAST_POS];

					// Version Classic
					///*
					TML_MTR_INST[i]._cfg.absFbk = 2;

					TML_MTR_INST[i]._cfg.HeartBeat = 0.4;
					TML_MTR_INST[i]._cfg.PVTPeriod = 0.08;

					//strcpy(TML_MTR_INST[i]._cfg.programName , "2023_BPV2_OSC_WRST.sw");
					//TML_MTR_INST[i].ProgramVersion = ASC2UDINT("2023");

					strcpy(TML_MTR_INST[i]._cfg.programName , "0344_BPV_WRST_OSC.sw");
					TML_MTR_INST[i].ProgramVersion = ASC2UDINT("0344");

					TML_MTR_INST[i].FirmwareVersion = ASC2UDINT("674C");  //0x674B
					TML_MTR_INST[i]._cfg.NotAutoDownload = 1;

					//TML_MTR_INST[i]._cfg.AnalLimitPos = 3900;
					//TML_MTR_INST[i]._cfg.AnalLimitNeg = 100;

					//TML_MTR_INST[i]._cfg.actPos2_scale = 70.0/4006.0;

					TML_MTR_INST[i]._cfg.AnalLimitPos = 0;
					TML_MTR_INST[i]._cfg.AnalLimitNeg = 0;

					TML_MTR_INST[i]._cfg.actPos2_scale = 0.0;

				break;

				case TML_AX_AVC:

					strcpy(TML_MTR_INST[i].Name , "AVC");

					// Analog Feedback from REF
					TML_MTR_INST[i]._cfg.loopPeriod = 0.001;
					TML_MTR_INST[i]._cfg.units = 4096;
					TML_MTR_INST[i]._cfg.rev_motor = 1;
					TML_MTR_INST[i]._cfg.rev_scale = 1.0/5.0;
					TML_MTR_INST[i]._cfg.maxVel = 1500.0;
					TML_MTR_INST[i]._cfg.maxAcc = TML_MTR_INST[i]._cfg.maxVel * 10.0;
					//TML_MTR_INST[i]._cfg.satpMax = 27853; // KPP bylo Stauration of proportional gain
					TML_MTR_INST[i]._cfg.satpMax = 32000; // KPP bylo Stauration of proportional gain
					//TML_MTR_INST[i]._cfg.kppMax = 32000; // KPP bylo Stauration of proportional gain
					//TML_MTR_INST[i]._cfg.kipMax = 200; // KPP bylo Stauration of proportional gain
					TML_MTR_INST[i]._cfg.kppMax = 32000;
					TML_MTR_INST[i]._cfg.kipMax = 1000;
					TML_MTR_INST[i]._cfg.absFbk = 0;

					TML_MTR_INST[i]._cfg.HeartBeat = 0.8;

					TML_MTR_INST[i]._cfg.signFilter = curCfg->Param[parAVC_FbkFilter].val[0];

					//U_BEND_HP_PINS
					strcpy(TML_MTR_INST[i]._cfg.programName , "0323_BPV_AVC.sw");
					TML_MTR_INST[i].ProgramVersion = ASC2UDINT("0323");

					TML_MTR_INST[i].FirmwareVersion = ASC2UDINT("6A2B");  //0x674C , 514D
					TML_MTR_INST[i]._cfg.Appl_ID_adr = 0x7FCF;
					TML_MTR_INST[i]._cfg.NotAutoDownload = 1;

					//TML_MTR_INST[i]._cfg.sftLimitPos = 0.0;
					//TML_MTR_INST[i]._cfg.sftLimitNeg = 0.0;

					/*
					TML_MTR_INST[i]._cfg.AnalLimitPos = 3900;
					TML_MTR_INST[i]._cfg.AnalLimitNeg = 100;
					*/

					TML_MTR_INST[i]._cfg.AnalLimitPos = 0;
					TML_MTR_INST[i]._cfg.AnalLimitNeg = 0;

				break;

				case TML_AX_WRST:

					strcpy(TML_MTR_INST[i].Name , "WRIST");

					// Analog Feedback from REF
					TML_MTR_INST[i]._cfg.loopPeriod = 0.001;

					TML_MTR_INST[i]._cfg.units = 1024 * 4;
					TML_MTR_INST[i]._cfg.rev_motor = -3.9 * 50 ;
					TML_MTR_INST[i]._cfg.rev_scale = -1.0/ (0.625 * 25.4 *M_PI) ;
					TML_MTR_INST[i]._cfg.maxVel = 8000.0/60.0/TML_MTR_INST[i]._cfg.rev_motor/ TML_MTR_INST[i]._cfg.rev_scale;
					TML_MTR_INST[i]._cfg.maxAcc = TML_MTR_INST[i]._cfg.maxVel * 10.0 ;
					TML_MTR_INST[i]._cfg.absLastPos = OLD_MTR_POS[WRST_LAST_POS];
					TML_MTR_INST[i]._cfg.absFbk = 2;

					TML_MTR_INST[i]._cfg.HeartBeat = 2.0;
					TML_MTR_INST[i]._cfg.PVTPeriod = 0.08;

					// Drive swap with OSC
					strcpy(TML_MTR_INST[i]._cfg.programName , "0322_BPV_OSC.sw");
					TML_MTR_INST[i].ProgramVersion = ASC2UDINT("0322");

					TML_MTR_INST[i].FirmwareVersion = ASC2UDINT("674C");  //0x674B
					TML_MTR_INST[i]._cfg.NotAutoDownload = 1;

					//TML_MTR_INST[i]._cfg.sftLimitPos = curCalib->Points[CALIB_OSC_SFT_LIMIT].val[0];
					//TML_MTR_INST[i]._cfg.sftLimitNeg = curCalib->Points[CALIB_OSC_SFT_LIMIT].val[1];

					//TML_MTR_INST[i]._cfg.sftLimitPos = 0.0;
					//TML_MTR_INST[i]._cfg.sftLimitNeg = 0.0;

				break;

				case TML_AX_WF:
				case TML_AX_WF_1:

					switch(i){

						case TML_AX_WF:

							strcpy(TML_MTR_INST[i].Name , "WF");
							TML_MTR_INST[i]._cfg.rev_scale = 1.0 /( 0.75 * 25.4 * M_PI) ;
							TML_MTR_INST[i]._cfg.rev_motor = 35.0;

						break;

						case TML_AX_WF_1:

							strcpy(TML_MTR_INST[i].Name , "WF_1");
							TML_MTR_INST[i]._cfg.rev_scale = -1.0 /( 0.75 * 25.4 * M_PI) ;
							TML_MTR_INST[i]._cfg.rev_motor = -35.0;

						break;

					}

					// Analog Feedback from REF
					TML_MTR_INST[i]._cfg.loopPeriod = 0.001;
					TML_MTR_INST[i]._cfg.units = 1024 * 4; //
					//TML_MTR_INST[i]._cfg.rev_motor = 35;

					TML_MTR_INST[i]._cfg.maxVel = 520 * 25.4/ 60.0; //// 520 ipm
					//TML_MTR_INST[i]._cfg.maxAcc = TML_MTR_INST[i]._cfg.maxVel * 100.0;
					TML_MTR_INST[i]._cfg.maxAcc = TML_MTR_INST[i]._cfg.maxVel * 4.0;
					TML_MTR_INST[i]._cfg.absFbk = 0;

					TML_MTR_INST[i]._cfg.HeartBeat = 0.4;

					strcpy(TML_MTR_INST[i]._cfg.programName , "0325_BPV_WF.sw");
					TML_MTR_INST[i].ProgramVersion = ASC2UDINT("0325");

					TML_MTR_INST[i].FirmwareVersion = ASC2UDINT("6A2B");
					TML_MTR_INST[i]._cfg.Appl_ID_adr = 0x7FCF;
					TML_MTR_INST[i]._cfg.NotAutoDownload = 1;

				break;

				case TML_AX_WP:
				case TML_AX_WP_1:

					switch(i){

						case TML_AX_WP: strcpy(TML_MTR_INST[i].Name , "WP"); break;
						case TML_AX_WP_1: strcpy(TML_MTR_INST[i].Name , "WP_1"); break;

					}

					// Analog Feedback from REF
					TML_MTR_INST[i]._cfg.loopPeriod = 0.001;

					TML_MTR_INST[i]._cfg.units = 500 * 4;
					TML_MTR_INST[i]._cfg.rev_motor = 24;
					TML_MTR_INST[i]._cfg.rev_scale = 1.0/5.0;
					TML_MTR_INST[i]._cfg.maxVel = 10000.0; //
					TML_MTR_INST[i]._cfg.maxAcc = 100.0;
					TML_MTR_INST[i]._cfg.absFbk = 0;

					TML_MTR_INST[i]._cfg.HeartBeat = 0.4;

					strcpy(TML_MTR_INST[i]._cfg.programName , "0326_BPV_WP.sw");
					TML_MTR_INST[i].ProgramVersion = ASC2UDINT("0326");

					TML_MTR_INST[i].FirmwareVersion = ASC2UDINT("6A2B");
					TML_MTR_INST[i]._cfg.Appl_ID_adr = 0x7FCF;
					TML_MTR_INST[i]._cfg.NotAutoDownload = 1;

				break;

				default:

					//strcpy(TML_MTR_INST[i].Name , "Spare ");
					xsprintf(TML_MTR_INST[i].Name, "Spare %d", i );

				break;

			}

		TML_MTR_INST[i].xCMD = TML_RESTART;

	}

		TML_mgr[0].hrdw[0].AxisNum = 0;
		TML_mgr[0].hrdw[1].AxisNum = 13;

		TML_mgr[0].pAxis[0] = &AxisCh[TML_mgr[0].hrdw[0].AxisNum];
		TML_mgr[0].pAxis[1] = &AxisCh[TML_mgr[0].hrdw[0].AxisNum];

		TML_mgr[0].pTML[0] = &TML_MTR_INST[0];
		TML_mgr[0].pTML[1] = &TML_MTR_INST[TML_mgr[0].hrdw[0].AxisNum];

		AxisCh[TML_AX_TVL].AxisID	= 1;
		//AxisCh[TML_AX_OSC].AxisID 	= 2;
		AxisCh[TML_AX_WRST].AxisID 	= 2;
		AxisCh[TML_AX_AVC].AxisID 	= 3;
		//AxisCh[TML_AX_WRST].AxisID 	= 4;
		AxisCh[TML_AX_OSC].AxisID 	= 4;

		AxisCh[TML_AX_WF].AxisID 	= 5;
		AxisCh[TML_AX_WP].AxisID 	= 6;
		AxisCh[TML_AX_WF_1].AxisID 	= 7;
		AxisCh[TML_AX_WP_1].AxisID 	= 8;
		/**************************************/
		/****   Process   ************************/

		// Lincoln Power Supply
		for(i=0 ; i < 1; i++){

			switch(i){

				case 0:

					strcpy(Process[PROC_TIG_PS].Name , "TIG PS");
					PS_Param_Set[i].pPrc = &Process[PROC_TIG_PS];

					PS_Param_Set[i].pCalibPoints		= &m->pCalib->Points[CALIB_TIG_AMPS_CMD];
					//PS_Param_Set[i].rawCmdMax			= 26170; // //
					//PS_Param_Set[i].AmpCMD_Max			= 500.0; // 62.5 amp / 1 V
					PS_Param_Set[i].rawCmdMax			= 32767;
					PS_Param_Set[i].AmpCMD_Max			= 627.0;

					PS_Param_Set[i].pArcLinkRobot   = (UDINT)&ArcLink.robot;

					//PS_Param_Set[i].Mode 			= 1; // Arclink connection

				break;

			}

		}
		///////////////////////////////////////////////////////

		for(i=0 ; i < 1 ; i++){

			switch(i){

				case 0:

					strcpy(Process[PROC_AVC].Name , "AVC");

					strcpy(VectorStateMach[VECT_AVC].Name , "AVC");

					AVC_Param_Set[i].pPrc = &Process[PROC_AVC];
					AVC_Param_Set[i].pVect = &VectorStateMach[VECT_AVC];
					AVC_Param_Set[i].VectStateNum = 1;
					AVC_Param_Set[i].Mode = 1; //BPV Mode
					AVC_Param_Set[i].MaxSpeedJog = TML_MTR_INST[TML_AX_AVC]._cfg.maxVel;

					m->pCalib->Points[CALIB_TIG_VOLT_FBK].num = 10;
					AVC_Param_Set[i].pCalibPoints		= &m->pCalib->Points[CALIB_TIG_VOLT_FBK];

				break;

			}
		}

		for(i=0 ; i < 1 ; i++){

			switch(i){

				case 0:

					strcpy(Process[m->pCfg->HeadCfg.WRST.PROC_Indx].Name , "WRST");
					strcpy(VectorStateMach[m->pCfg->HeadCfg.WRST.VECT_A_Indx].Name , "WRST");

					WRST_TML_Param_Set[i].pPrc = &Process[m->pCfg->HeadCfg.WRST.PROC_Indx];
					WRST_TML_Param_Set[i].pVect = &VectorStateMach[m->pCfg->HeadCfg.WRST.VECT_A_Indx];
					WRST_TML_Param_Set[i].VectStateNum = 1;
					WRST_TML_Param_Set[i].pTML = &TML_MTR_INST[m->pCfg->HeadCfg.WRST.TML_A_Indx] ;
					WRST_TML_Param_Set[i].Mode = 0;

					WRST_TML_Param_Set[i].GlbDirection = 1.0;

					WRST_TML_Param_Set[i].MaxAmpl = 0.0;

				break;

			}
		}

		for(i=0 ; i < 1 ; i++){

			switch(i){

				case 0:

					strcpy(Process[PROC_OSC].Name , "OSC");
					strcpy(VectorStateMach[VECT_OSC].Name , "OSC");

					/* Tak bylo we Flange
					OSC_TML_Param_Set[i].pPrc = &Process[PROC_OSC];
					OSC_TML_Param_Set[i].pVect = &VectorStateMach[VECT_OSC];
					OSC_TML_Param_Set[i].VectStateNum = 1;
					OSC_TML_Param_Set[i].pTML = &TML_MTR_INST[TML_AX_OSC] ;

					OSC_TML_Param_Set[i].Mode = 3; // Exp BEMF
					OSC_TML_Param_Set[i].PosFbkIndx = 2;

					////  New Oscillation concept - BEMF
					//OSC_TML_Param_Set[i].mm2ticks = TML_MTR_INST[TML_AX_OSC]._cfg.units * TML_MTR_INST[TML_AX_OSC]._cfg.rev_scale;
					OSC_TML_Param_Set[i].mm2ticks = 4096.0/80.0;
					//OSC_TML_Param_Set[i].SpeedFactor = 410;
					//OSC_TML_Param_Set[i].MaxOscAmpl = 1.0 * 25.4;
					OSC_TML_Param_Set[i].MaxOscAmpl = 0.0;

					OSC_TML_Param_Set[i].SpeedFactor = 10.0;
					*/
					////////////

					OSC_TML_Param_Set[i].pPrc = &Process[PROC_OSC];
					OSC_TML_Param_Set[i].pVect = &VectorStateMach[VECT_OSC];
					OSC_TML_Param_Set[i].VectStateNum = 1;
					OSC_TML_Param_Set[i].pTML = &TML_MTR_INST[TML_AX_OSC] ;

					OSC_TML_Param_Set[i].Mode = 1; //BPV Mode
					OSC_TML_Param_Set[i].MaxOscAmpl = 0.0;

					////////////////////////////////////////////////

				break;

			}

		}

		for(i=0 ; i < 1 ; i++){

			switch(i){

				case 0:

					strcpy(Process[PROC_GAS].Name , "GAS");
					GAS_Param_Set[i].pPrc = &Process[PROC_GAS];

					GAS_Param_Set[i].pSensInput     = &Hardware[1].Inp[5];  //FourAxis Head
					GAS_Param_Set[i].pOutput		= &Hardware[1].Outp[4];

				break;

			}

		}

		for(i=0 ; i < 1 ; i++){

			switch(i){

				case 0:

					strcpy(Process[m->pCfg->HeadCfg.INDX.PROC_Indx].Name , "INDX");
					INDEX_Param_Set[i].pPrc = &Process[m->pCfg->HeadCfg.INDX.PROC_Indx];
					//INDEX_Param_Set[i].pPrc = &Process[PROC_INDX];
					INDEX_Param_Set[i].pVect = &VectorStateMach[m->pCfg->HeadCfg.INDX.VECT_A_Indx];
					strcpy(VectorStateMach[m->pCfg->HeadCfg.INDX.VECT_A_Indx].Name , "INDX A");
					strcpy(VectorStateMach[m->pCfg->HeadCfg.INDX.VECT_B_Indx].Name , "INDX B");
					INDEX_Param_Set[i].VectStateNum = 2;
					INDEX_Param_Set[i].Mode = 0;
					INDEX_Param_Set[i].MaxSpeed = 24.0;
					INDEX_Param_Set[i].pCalibPoints		= &m->pCalib->Points[CALIB_TIG_AMPS_CMD];

				break;

			}

		}

		for(i=0 ; i < 1; i++){

			switch(i){

				case 0:

					strcpy(Process[PROC_COOL].Name , "COOLANT");
					COOL_Param_Set[i].pPrc = &Process[PROC_COOL];

					COOL_Param_Set[i].pSensInput     = &Hardware[1].Inp[4];  //FourAxis Head
					COOL_Param_Set[i].pOutput		= &Hardware[1].Outp[6];

				break;

			}

		}

		for(i=0 ; i < 1; i++){

			switch(i){

				case 0:

					strcpy(Process[PROC_HW_PS].Name , "HW PS");
					HW_PS_Param_Set[i].pPrc = &Process[PROC_HW_PS];

					HW_PS_Param_Set[i].pCalibPoints		= &m->pCalib->Points[CALIB_HW_AMPS_CMD];
					HW_PS_Param_Set[i].rawCmdMax 		= 16383.0;
					HW_PS_Param_Set[i].AmpCMD_Max 		= 160.0;

				break;

			}

		}

		for(i=0 ; i < 2; i++){

			switch(i){

				case 0:

					strcpy(Process[PROC_WIRE_FEED].Name ,"WrFeed");
					strcpy(VectorStateMach[VECT_WF].Name ,"WrFeed#1");
					strcpy(VectorStateMach[VECT_WF_1].Name ,"WrFeed#2");

					WIRE_Param_Set[i].pPrc = &Process[PROC_WIRE_FEED];
					WIRE_Param_Set[i].pVect = &VectorStateMach[VECT_WF];
					WIRE_Param_Set[i].VectStateNum = 1; //BPV Mode
					WIRE_Param_Set[i].Mode = 1;
					WIRE_Param_Set[i].MaxSpeedJog = TML_MTR_INST[TML_AX_WF]._cfg.maxVel;

					WIRE_Param_Set[i].pSynchMode = &WFSynchMode;
					WIRE_Param_Set[i].pSynchClock = &SynchClckToWF;

					WIRE_Param_Set[i].pCalibPoints	= &m->pCalib->Points[CALIB_WF_SPEED_CMD];

				break;

				case 1:

					strcpy(Process[PROC_WIRE_PULSE].Name ,"WrPulse");
					strcpy(VectorStateMach[VECT_WP].Name ,"WrPulse#1");
					strcpy(VectorStateMach[VECT_WP_1].Name ,"WrPulse#2");
					WIRE_Param_Set[i].Mode = 1; //BPV Mode

					WIRE_Param_Set[i].pPrc = &Process[PROC_WIRE_PULSE];
					WIRE_Param_Set[i].pVect = &VectorStateMach[VECT_WP];
					WIRE_Param_Set[i].VectStateNum = 1;

					WIRE_Param_Set[i].pSynchMode = &WPSynchMode;
					WIRE_Param_Set[i].pSynchClock = &SynchClckToWP;

					WIRE_Param_Set[i].pCalibPoints	= &m->pCalib->Points[CALIB_WP_SPEED_CMD];

				break;

		}

		}

		for(i=0 ; i < 1; i++){

			switch(i){

				case 0:

					strcpy(Process[PROC_TVL].Name , "TVL");
					strcpy(VectorStateMach[VECT_TVL].Name , "TVL");

					TVL_ROT_Param_Set[i].Mode = 1; //BPV Mode
					TVL_ROT_Param_Set[i].MaxSpeedJog = TML_MTR_INST[TML_AX_TVL]._cfg.maxVel;

					TVL_ROT_Param_Set[i].pPrc = &Process[PROC_TVL];
					TVL_ROT_Param_Set[i].pVect = &VectorStateMach[VECT_TVL];
					TVL_ROT_Param_Set[i].VectStateNum = 1;

					TVL_ROT_Param_Set[i].VectModeForJog = vectSt_Mode_Volt;

					TVL_ROT_Param_Set[i].TotalRescaleFactor = 1.0;
					TVL_ROT_Param_Set[i].pCalibPoints = &m->pCalib->Points[CALIB_TVL_SPEED_CMD];

					TVL_ROT_Param_Set[i].pTrackDia = &curCfg->Param[parTVL_TrackDia].val[0];
					TVL_ROT_Param_Set[i].pVelTolerance = &curCfg->Param[parTVL_SpeedTolerane].val[0];

					// TVL in Torq Mode
					TVL_ROT_Param_Set[i].VectModeForJog = vectSt_Mode_Vel;

					TVL_ROT_Param_Set[i].pEncoder = &AxisCh[TML_AX_TVL].curPos;
					TVL_ROT_Param_Set[i].pHomePos = &OLD_MTR_POS[TVL_ENC_HOME];
					TVL_ROT_Param_Set[i].EncPerTick = m->pCfg->HeadCfg.TVL.EncPerTick;
					TVL_ROT_Param_Set[i].EncDir = m->pCfg->HeadCfg.TVL.Enc_Dir;
					TVL_ROT_Param_Set[i].TicksAtHighVel = 20;

					TVL_ROT_Param_Set[i].pSynchMode = &TVLSynchMode;
					TVL_ROT_Param_Set[i].pSynchClock = &SynchClckToTVL;

			break;

	}

	}

	////////////////////////////////////////////
	/*
	Process[PROC_OSC].Disable = 1;
	Process[PROC_OSC].TestMode = 1;
	VectorStateMach[VECT_OSC].simul = 1;
	TML_MTR_INST[TML_AX_OSC].Disable = 1;
	*/

	Process[PROC_WRST].Disable = 0;
	Process[PROC_WRST].TestMode = 0;
	VectorStateMach[VECT_WRST].simul = 0;
	TML_MTR_INST[TML_AX_WRST].Disable = 0;

	////////////////////////////////////////////////////////////
	/// To jest Tylko do proby
	/*
	VectorStateMach[VECT_AVC].simul = 1;
	VectorStateMach[VECT_OSC].simul = 1;
	VectorStateMach[VECT_TVL].simul = 1;
	VectorStateMach[VECT_INDX_1].simul = 1;
	VectorStateMach[VECT_INDX_2].simul = 1;
	VectorStateMach[VECT_WF_1].simul = 1;
	VectorStateMach[VECT_WF].simul = 1;
	VectorStateMach[VECT_WP_1].simul = 1;
	VectorStateMach[VECT_WP].simul = 1;

	VectorStateMach[VECT_AVC].testMode = 1;
	VectorStateMach[VECT_OSC].testMode = 1;
	VectorStateMach[VECT_TVL].testMode = 1;
	VectorStateMach[VECT_INDX_1].testMode = 1;
	VectorStateMach[VECT_INDX_2].testMode = 1;
	VectorStateMach[VECT_WF_1].testMode = 1;
	VectorStateMach[VECT_WF].testMode = 1;
	VectorStateMach[VECT_WP_1].testMode = 1;
	VectorStateMach[VECT_WP].testMode = 1;

	// To tylko trzeba uncomment gdy jest bez torch ale reszta dziala
	TML_MTR_INST[TML_AX_AVC].Disable = 1;
	TML_MTR_INST[TML_AX_OSC].Disable = 1;
	TML_MTR_INST[TML_AX_TVL].Disable = 1;
	TML_MTR_INST[TML_AX_WRST].Disable = 1;
	TML_MTR_INST[TML_AX_WF].Disable = 1;
	TML_MTR_INST[TML_AX_WF_1].Disable = 1;
	TML_MTR_INST[TML_AX_WP].Disable = 1;
	TML_MTR_INST[TML_AX_WP_1].Disable = 1;
	////////////////////////////////////////

	Process[PROC_AVC].Disable = 1;
	Process[PROC_AVC].TestMode = 1;

	Process[PROC_INDX].Disable = 1;
	Process[PROC_INDX].TestMode = 1;

	Process[PROC_OSC].Disable = 1;
	Process[PROC_OSC].TestMode = 1;

	Process[PROC_TVL].Disable = 1;
	Process[PROC_TVL].TestMode = 1;

	Process[PROC_WIRE_FEED].Disable = 1;
	Process[PROC_WIRE_FEED].TestMode = 1;

	Process[PROC_WIRE_PULSE].Disable = 1;
	Process[PROC_WIRE_PULSE].TestMode = 1;

	Process[PROC_COOL].Disable = 1;
	Process[PROC_COOL].TestMode = 1;

	Process[PROC_GAS].Disable = 1;
	Process[PROC_GAS].TestMode = 1;
	*/
	////////////////////////////////////////////////////////

	return 1;

}

DINT Configure_BPV_F_HEAD(MASTER_typ * m, UINT headType){
int i;

CurCfg_typ *curCfg;
Cfg_typ *cfg;
CurCalib_typ *curCalib , *defaultCalib;

	if(!m)
		return;

	curCfg = (CurCfg_typ*)m->pCurCfg;
	cfg = (Cfg_typ*)m->pCfg;

	curCalib = m->pCalib;
	defaultCalib = m->pDefaultCalib;

	if(!curCfg || !cfg || !curCalib  || !defaultCalib)
		return;

/*********************************************/
	/***   Hardware and Vectors *********************/

	TML_MTR_INST[m->pCfg->HeadCfg.TVL.TML_Indx ].pState = &VectorStateMach[m->pCfg->HeadCfg.TVL.VECT_Indx];

	TML_MTR_INST[m->pCfg->HeadCfg.AVC.TML_A_Indx ].pState = &VectorStateMach[m->pCfg->HeadCfg.AVC.VECT_A_Indx];
	TML_MTR_INST[m->pCfg->HeadCfg.AVC.TML_B_Indx ].pState = &VectorStateMach[m->pCfg->HeadCfg.AVC.VECT_B_Indx];

	TML_MTR_INST[m->pCfg->HeadCfg.OSC.TML_A_Indx ].pState = &VectorStateMach[m->pCfg->HeadCfg.OSC.VECT_A_Indx];
	TML_MTR_INST[m->pCfg->HeadCfg.OSC.TML_B_Indx ].pState = &VectorStateMach[m->pCfg->HeadCfg.OSC.VECT_B_Indx];

	TML_MTR_INST[m->pCfg->HeadCfg.WF.TML_A_Indx ].pState = &VectorStateMach[m->pCfg->HeadCfg.WF.VECT_A_Indx];
	TML_MTR_INST[m->pCfg->HeadCfg.WF.TML_B_Indx ].pState = &VectorStateMach[m->pCfg->HeadCfg.WF.VECT_B_Indx];

	TML_MTR_INST[m->pCfg->HeadCfg.WP.TML_A_Indx ].pState = &VectorStateMach[m->pCfg->HeadCfg.WP.VECT_A_Indx];
	TML_MTR_INST[m->pCfg->HeadCfg.WP.TML_B_Indx ].pState = &VectorStateMach[m->pCfg->HeadCfg.WP.VECT_B_Indx];

	TML_MTR_INST[m->pCfg->HeadCfg.WRST.TML_A_Indx ].pState = &VectorStateMach[m->pCfg->HeadCfg.WRST.VECT_A_Indx];
	TML_MTR_INST[m->pCfg->HeadCfg.WRST.TML_B_Indx ].pState = &VectorStateMach[m->pCfg->HeadCfg.WRST.VECT_B_Indx];

	DC_Mtr[m->pCfg->HeadCfg.INDX.DC_A_Indx ].pState = &VectorStateMach[m->pCfg->HeadCfg.INDX.VECT_A_Indx];
	DC_Mtr[m->pCfg->HeadCfg.INDX.DC_B_Indx ].pState = &VectorStateMach[m->pCfg->HeadCfg.INDX.VECT_B_Indx];

	/*********************************************************/
	/****   Phisical hardware configuration   ************************/

		for(i = 0 ; i < PROCESS_NUM; i++)
			strcpy(Process[i].Name , "spare");

		for(i = 0 ; i < VECTORS_NUM; i++)
			strcpy(VectorStateMach[i].Name , "spare");

			/***********************************/

		//////////////////////////////////////////////////////////////////////////////////
		// Wire Block
		for(i=0 ; i < 2; i++){

			switch(i){

				case 0:
					strcpy(Process[m->pCfg->HeadCfg.WB[i].PROC_Indx].Name , "WB_UD");
					strcpy(VectorStateMach[m->pCfg->HeadCfg.WB[i].VECT_Indx].Name , "WB_UD");

					WR_BLK_Param_Set[i].pPrc = &Process[m->pCfg->HeadCfg.WB[i].PROC_Indx];
					WR_BLK_Param_Set[i].pVect = &VectorStateMach[m->pCfg->HeadCfg.WB[i].VECT_Indx];
					WR_BLK_Param_Set[i].VectStateNum = 1;

					WR_BLK_Param_Set[i].MaxSpeedJog = 24.0;

					Gen_one = 1.0;
					WR_BLK_Param_Set[i].pJogSpeed = &Gen_one;

				break;

				case 1:
					strcpy(Process[m->pCfg->HeadCfg.WB[i].PROC_Indx].Name , "WB_LR");
					strcpy(VectorStateMach[m->pCfg->HeadCfg.WB[i].VECT_Indx].Name , "WB_LR");

					WR_BLK_Param_Set[i].pPrc = &Process[PROC_WB_LR];
					WR_BLK_Param_Set[i].pVect = &VectorStateMach[VECT_WB_LR];
					WR_BLK_Param_Set[i].VectStateNum = 1;

					WR_BLK_Param_Set[i].MaxSpeedJog = 24.0;

					Gen_one = 1.0;
					WR_BLK_Param_Set[i].pJogSpeed = &Gen_one;

				break;

			}

		}

		for(i = 0 ; i < DC2DIRMTR_NUM; i++){

			switch(i){

				case DC_WB_UD:

					strcpy(DC2DirMtr[i].Name , "WB_UD");
					DC2DirMtr[i].pState = &VectorStateMach[VECT_WB_UD];

					DC2DirMtr[i].Cfg.pQ1_output = &Hardware[1].Outp[12];
					DC2DirMtr[i].Cfg.pQ2_output = &Hardware[1].Outp[13];
					DC2DirMtr[i].Cfg.pQ3_output = &Hardware[1].Outp[14];
					DC2DirMtr[i].Cfg.pQ4_output = &Hardware[1].Outp[15];

					DC2DirMtr[i].Cfg.MtrDir = 1.0;

				break;

				case DC_WB_LR:

					strcpy(DC2DirMtr[i].Name , "WB_LR");
					DC2DirMtr[i].pState = &VectorStateMach[VECT_WB_LR];

					DC2DirMtr[i].Cfg.pQ1_output = &Hardware[1].Outp[16];
					DC2DirMtr[i].Cfg.pQ2_output = &Hardware[1].Outp[17];
					DC2DirMtr[i].Cfg.pQ3_output = &Hardware[1].Outp[18];
					DC2DirMtr[i].Cfg.pQ4_output = &Hardware[1].Outp[19];

					DC2DirMtr[i].Cfg.MtrDir = 1.0;

				break;

			}

		}
		/////////////////////////////////////////////////////////////////////////////////

		for(i = 0 ; i < GEN_MTR_NUM; i++){

			switch(i){

				case DC_INDX_1:
				case DC_INDX_2:

					switch(i){

						case DC_INDX_1:

							strcpy(DC_Mtr[i].Name , "DC INDX #1");

							DC_Mtr[i].Cfg.mtr_dir = 1.0;

							if(ProjectConfig == project_US_Orbital) // US Orbital has B and /B swapped
								DC_Mtr[i].Cfg.enc_dir = 1.0;
							else
								DC_Mtr[i].Cfg.enc_dir = -1.0;

							//DC_Mtr[i].Cfg.enc_dir = -1.0;

						break;

						case DC_INDX_2:

							strcpy(DC_Mtr[i].Name , "DC INDX #2");

							DC_Mtr[i].Cfg.mtr_dir = -1.0;

							if(ProjectConfig == project_US_Orbital) // US Orbital has B and /B swapped
								DC_Mtr[i].Cfg.enc_dir = -1.0;
							else
								DC_Mtr[i].Cfg.enc_dir = 1.0;

							//DC_Mtr[i].Cfg.enc_dir = 1.0;

						break;

					}

					//DC_Mtr[i].Cfg.units = 2000 / 59.847340050885561192713356451475; // 2000 enc ticks / 0.75 " dia * 25.4 * PI
					//DC_Mtr[i].Cfg.rev_scale = 66.0 * 0.218686666; // Ratio gear box 66:1

					DC_Mtr[i].Cfg.units =48000 / (1.25 * M_PI * 25.4); // 48000 enc ticks / 1.25 " dia * 25.4 * PI
					DC_Mtr[i].Cfg.rev_scale = 1; // Ratio gear box 66:1

					/* Parameters for PID controller */
					// To nowe
					DC_Mtr[i].msc.PIDParameters.Kp= 100.0;//0.4; //proportional gain / was 0.6
					DC_Mtr[i].msc.PIDParameters.Tn= 0.0;//0.3.1; //intergral action time
					DC_Mtr[i].msc.PIDParameters.Kfbk = 0.1; //windup dampenin

					DC_Mtr[i].msc.PID.enable = 0;
					DC_Mtr[i].msc.PID.pPar = &DC_Mtr[i].msc.PIDParameters;
					DC_Mtr[i].msc.PID.request = 3; // Read parameters from PIDParameters
					DC_Mtr[i].msc.PIDParameters.Tv= 0; //derivative action time
					DC_Mtr[i].msc.PIDParameters.Y_max = 100.0;	//max manipulated variable %
					DC_Mtr[i].msc.PIDParameters.Y_min = -100.0; //min manipulated variable %

				break;

				default:

					strcpy(DC_Mtr[i].Name , "Spare ");

				break;

			}

				//CalcUnits(&DC_Mtr[i]);
				DC_Mtr[i].msc.kPos = (float)DC_Mtr[i].Cfg.units * DC_Mtr[i].Cfg.rev_scale;

		}

		for(i = 0 ; i < TML_SERVO_NUM ; i++){

			switch(i){

				case TML_AX_TVL:

					strcpy(TML_MTR_INST[i].Name , "TVL");

					TML_MTR_INST[i]._cfg.loopPeriod = 0.0005; // Slow loop
					TML_MTR_INST[i]._cfg.units = 1024 * 4; //
					TML_MTR_INST[i]._cfg.rev_motor = 156;
					TML_MTR_INST[i]._cfg.rev_scale = 1.0 /( 1.25 * 25.4 * M_PI) ;

					TML_MTR_INST[i]._cfg.maxVel =  4500.0/60.0/TML_MTR_INST[i]._cfg.rev_motor/ TML_MTR_INST[i]._cfg.rev_scale;
					TML_MTR_INST[i]._cfg.maxAcc = TML_MTR_INST[i]._cfg.maxVel * 10.0 ;
					TML_MTR_INST[i]._cfg.absLastPos = OLD_MTR_POS[TVL_LAST_POS];
					TML_MTR_INST[i]._cfg.absFbk = 2;

					TML_MTR_INST[i]._cfg.HeartBeat = 0.08;

					strcpy(TML_MTR_INST[i]._cfg.programName , "0331_BPV_TVL.sw");
					TML_MTR_INST[i].ProgramVersion = ASC2UDINT("0331");

					TML_MTR_INST[i].FirmwareVersion = ASC2UDINT("6A2B");  //0x674B
					TML_MTR_INST[i]._cfg.Appl_ID_adr = 0x7FCF;
					TML_MTR_INST[i]._cfg.NotAutoDownload = 1;

				break;

				case TML_AX_OSC:

					strcpy(TML_MTR_INST[i].Name , "OSC");

					// Analog Feedback from REF
					TML_MTR_INST[i]._cfg.loopPeriod = 0.001;

					TML_MTR_INST[i]._cfg.units = 1024 * 4;
					//TML_MTR_INST[i]._cfg.rev_motor = -3.9 * 50 ;
					TML_MTR_INST[i]._cfg.rev_motor = (-75.0/19.0) * 50.0;
					TML_MTR_INST[i]._cfg.rev_scale = -1.0/ (0.625 * 25.4 *M_PI) ;

					TML_MTR_INST[i]._cfg.maxVel = 8000.0/60.0/TML_MTR_INST[i]._cfg.rev_motor/ TML_MTR_INST[i]._cfg.rev_scale;
					TML_MTR_INST[i]._cfg.maxAcc = TML_MTR_INST[i]._cfg.maxVel * 10.0 ;
					TML_MTR_INST[i]._cfg.absLastPos = OLD_MTR_POS[OSC_LAST_POS];
					TML_MTR_INST[i]._cfg.absFbk = 2;

					TML_MTR_INST[i]._cfg.HeartBeat = 0.4;
					TML_MTR_INST[i]._cfg.PVTPeriod = 0.08;

					// U_BEND_HP_PINS
					strcpy(TML_MTR_INST[i]._cfg.programName , "0322_BPV_OSC.sw");
					TML_MTR_INST[i].ProgramVersion = ASC2UDINT("0322");

					TML_MTR_INST[i].FirmwareVersion = ASC2UDINT("674C");  //0x674B
					TML_MTR_INST[i]._cfg.NotAutoDownload = 1;

					//TML_MTR_INST[i]._cfg.sftLimitPos = curCalib->Points[CALIB_OSC_SFT_LIMIT].val[0];
					//TML_MTR_INST[i]._cfg.sftLimitNeg = curCalib->Points[CALIB_OSC_SFT_LIMIT].val[1];

					//TML_MTR_INST[i]._cfg.sftLimitPos = 0.0;
					//TML_MTR_INST[i]._cfg.sftLimitNeg = 0.0;

				break;

				case TML_AX_AVC:
				case TML_AX_AVC2:

					if(i == TML_AX_AVC)
						strcpy(TML_MTR_INST[i].Name , "AVC");
					else
						strcpy(TML_MTR_INST[i].Name , "AVC_2");

					// Analog Feedback from REF
					TML_MTR_INST[i]._cfg.loopPeriod = 0.001;
					TML_MTR_INST[i]._cfg.units = 4096;
					TML_MTR_INST[i]._cfg.rev_motor = 1;
					TML_MTR_INST[i]._cfg.rev_scale = 1.0/5.0;
					TML_MTR_INST[i]._cfg.maxVel = 1500.0;
					TML_MTR_INST[i]._cfg.maxAcc = TML_MTR_INST[i]._cfg.maxVel * 10.0;
					//TML_MTR_INST[i]._cfg.satpMax = 27853; // KPP bylo Stauration of proportional gain
					TML_MTR_INST[i]._cfg.satpMax = 32000; // KPP bylo Stauration of proportional gain
					//TML_MTR_INST[i]._cfg.kppMax = 32000; // KPP bylo Stauration of proportional gain
					//TML_MTR_INST[i]._cfg.kipMax = 200; // KPP bylo Stauration of proportional gain
					TML_MTR_INST[i]._cfg.kppMax = 32000;
					TML_MTR_INST[i]._cfg.kipMax = 1000;
					TML_MTR_INST[i]._cfg.absFbk = 0;

					TML_MTR_INST[i]._cfg.HeartBeat = 0.8;

					TML_MTR_INST[i]._cfg.signFilter = curCfg->Param[parAVC_FbkFilter].val[0];

					//U_BEND_HP_PINS
					strcpy(TML_MTR_INST[i]._cfg.programName , "0323_BPV_AVC.sw");
					TML_MTR_INST[i].ProgramVersion = ASC2UDINT("0323");

					TML_MTR_INST[i].FirmwareVersion = ASC2UDINT("6A2B");  //0x674C , 514D
					TML_MTR_INST[i]._cfg.Appl_ID_adr = 0x7FCF;
					TML_MTR_INST[i]._cfg.NotAutoDownload = 1;

					//TML_MTR_INST[i]._cfg.sftLimitPos = 0.0;
					//TML_MTR_INST[i]._cfg.sftLimitNeg = 0.0;

					/*
					TML_MTR_INST[i]._cfg.AnalLimitPos = 3900;
					TML_MTR_INST[i]._cfg.AnalLimitNeg = 100;
					*/

					TML_MTR_INST[i]._cfg.AnalLimitPos = 0;
					TML_MTR_INST[i]._cfg.AnalLimitNeg = 0;

				break;

				case TML_AX_WRST:

					strcpy(TML_MTR_INST[i].Name , "WRIST");

					// Analog Feedback from REF
					TML_MTR_INST[i]._cfg.loopPeriod = 0.001;

					TML_MTR_INST[i]._cfg.units = 1024 * 4;
					TML_MTR_INST[i]._cfg.rev_motor = -3.9 * 50 ;
					TML_MTR_INST[i]._cfg.rev_scale = -1.0/ (0.625 * 25.4 *M_PI) ;
					TML_MTR_INST[i]._cfg.maxVel = 8000.0/60.0/TML_MTR_INST[i]._cfg.rev_motor/ TML_MTR_INST[i]._cfg.rev_scale;
					TML_MTR_INST[i]._cfg.maxAcc = TML_MTR_INST[i]._cfg.maxVel * 10.0 ;
					TML_MTR_INST[i]._cfg.absLastPos = OLD_MTR_POS[WRST_LAST_POS];
					TML_MTR_INST[i]._cfg.absFbk = 2;

					//TML_MTR_INST[i]._cfg.HeartBeat = 2.0;
					TML_MTR_INST[i]._cfg.PVTPeriod = 0.08;

					// U_BEND_HP_PINS
					//strcpy(TML_MTR_INST[i]._cfg.programName , "0334_BPV_WRST.sw");
					//TML_MTR_INST[i].ProgramVersion = ASC2UDINT("0334");

					//strcpy(TML_MTR_INST[i]._cfg.programName , "0344_BPV_WRST_OSC.sw");
					//TML_MTR_INST[i].ProgramVersion = ASC2UDINT("0344");

					strcpy(TML_MTR_INST[i]._cfg.programName , "0354_BPV_WRST_OSC_POT.sw");
					TML_MTR_INST[i].ProgramVersion = ASC2UDINT("0354");

					TML_MTR_INST[i].FirmwareVersion = ASC2UDINT("674C");  //0x674B
					//TML_MTR_INST[i]._cfg.NotAutoDownload = 1;
					TML_MTR_INST[i]._cfg.NotAutoDownload = 0;

					//TML_MTR_INST[i]._cfg.sftLimitPos = curCalib->Points[CALIB_OSC_SFT_LIMIT].val[0];
					//TML_MTR_INST[i]._cfg.sftLimitNeg = curCalib->Points[CALIB_OSC_SFT_LIMIT].val[1];

					//TML_MTR_INST[i]._cfg.sftLimitPos = 0.0;
					//TML_MTR_INST[i]._cfg.sftLimitNeg = 0.0;

				break;

				case TML_AX_WF:
				case TML_AX_WF_1:

					switch(i){

						case TML_AX_WF:

							strcpy(TML_MTR_INST[i].Name , "WF");
							TML_MTR_INST[i]._cfg.rev_scale = 1.0 /( 0.75 * 25.4 * M_PI) ;
							TML_MTR_INST[i]._cfg.rev_motor = 35.0;

						break;

						case TML_AX_WF_1:

							strcpy(TML_MTR_INST[i].Name , "WF_1");
							TML_MTR_INST[i]._cfg.rev_scale = -1.0 /( 0.75 * 25.4 * M_PI) ;
							TML_MTR_INST[i]._cfg.rev_motor = -35.0;

						break;

					}

					// Analog Feedback from REF
					TML_MTR_INST[i]._cfg.loopPeriod = 0.001;
					TML_MTR_INST[i]._cfg.units = 1024 * 4; //
					//TML_MTR_INST[i]._cfg.rev_motor = 35;

					TML_MTR_INST[i]._cfg.maxVel = 520 * 25.4/ 60.0; //// 520 ipm
					//TML_MTR_INST[i]._cfg.maxAcc = TML_MTR_INST[i]._cfg.maxVel * 100.0;
					TML_MTR_INST[i]._cfg.maxAcc = TML_MTR_INST[i]._cfg.maxVel * 4.0;
					TML_MTR_INST[i]._cfg.absFbk = 0;

					TML_MTR_INST[i]._cfg.HeartBeat = 0.4;

					strcpy(TML_MTR_INST[i]._cfg.programName , "0325_BPV_WF.sw");
					TML_MTR_INST[i].ProgramVersion = ASC2UDINT("0325");

					TML_MTR_INST[i].FirmwareVersion = ASC2UDINT("6A2B");
					TML_MTR_INST[i]._cfg.Appl_ID_adr = 0x7FCF;
					TML_MTR_INST[i]._cfg.NotAutoDownload = 1;

				break;

				case TML_AX_WP:
				case TML_AX_WP_1:

					switch(i){

						case TML_AX_WP: strcpy(TML_MTR_INST[i].Name , "WP"); break;
						case TML_AX_WP_1: strcpy(TML_MTR_INST[i].Name , "WP_1"); break;

					}

					// Analog Feedback from REF
					TML_MTR_INST[i]._cfg.loopPeriod = 0.001;

					TML_MTR_INST[i]._cfg.units = 500 * 4;
					TML_MTR_INST[i]._cfg.rev_motor = 24;
					TML_MTR_INST[i]._cfg.rev_scale = 1.0/5.0;
					TML_MTR_INST[i]._cfg.maxVel = 10000.0; //
					TML_MTR_INST[i]._cfg.maxAcc = 100.0;
					TML_MTR_INST[i]._cfg.absFbk = 0;

					TML_MTR_INST[i]._cfg.HeartBeat = 0.4;

					strcpy(TML_MTR_INST[i]._cfg.programName , "0326_BPV_WP.sw");
					TML_MTR_INST[i].ProgramVersion = ASC2UDINT("0326");

					TML_MTR_INST[i].FirmwareVersion = ASC2UDINT("6A2B");
					TML_MTR_INST[i]._cfg.Appl_ID_adr = 0x7FCF;
					TML_MTR_INST[i]._cfg.NotAutoDownload = 1;

				break;

				default:

					//strcpy(TML_MTR_INST[i].Name , "Spare ");
					xsprintf(TML_MTR_INST[i].Name, "Spare %d", i );

				break;

			}

		TML_MTR_INST[i].xCMD = TML_RESTART;

	}

		TML_mgr[0].hrdw[0].AxisNum = 0;
		TML_mgr[0].hrdw[1].AxisNum = 13;

		TML_mgr[0].pAxis[0] = &AxisCh[TML_mgr[0].hrdw[0].AxisNum];
		TML_mgr[0].pAxis[1] = &AxisCh[TML_mgr[0].hrdw[0].AxisNum];

		TML_mgr[0].pTML[0] = &TML_MTR_INST[0];
		TML_mgr[0].pTML[1] = &TML_MTR_INST[TML_mgr[0].hrdw[0].AxisNum];

		AxisCh[TML_AX_TVL].AxisID	= 1;
		AxisCh[TML_AX_OSC].AxisID 	= 2;
		//AxisCh[TML_AX_WRST].AxisID 	= 2;
		AxisCh[TML_AX_AVC].AxisID 	= 3;
		AxisCh[TML_AX_WRST].AxisID 	= 4;
		//AxisCh[TML_AX_OSC].AxisID 	= 4;

		AxisCh[TML_AX_WF].AxisID 	= 5;
		AxisCh[TML_AX_WP].AxisID 	= 6;
		AxisCh[TML_AX_WF_1].AxisID 	= 7;
		AxisCh[TML_AX_WP_1].AxisID 	= 8;
		/**************************************/
		/****   Process   ************************/

		// Lincoln Power Supply
		for(i=0 ; i < 1; i++){

			switch(i){

				case 0:

					strcpy(Process[PROC_TIG_PS].Name , "TIG PS");
					PS_Param_Set[i].pPrc = &Process[PROC_TIG_PS];

					PS_Param_Set[i].pCalibPoints		= &m->pCalib->Points[CALIB_TIG_AMPS_CMD];
					//PS_Param_Set[i].rawCmdMax			= 26170; // //
					//PS_Param_Set[i].AmpCMD_Max			= 500.0; // 62.5 amp / 1 V
					PS_Param_Set[i].rawCmdMax			= 32767;
					PS_Param_Set[i].AmpCMD_Max			= 627.0;

					PS_Param_Set[i].pArcLinkRobot   = (UDINT)&ArcLink.robot;

					//PS_Param_Set[i].Mode 			= 1; // Arclink connection

				break;

			}

		}
		///////////////////////////////////////////////////////

		for(i=0 ; i < 1 ; i++){

			switch(i){

				case 0:

					strcpy(Process[PROC_AVC].Name , "AVC");

					strcpy(VectorStateMach[VECT_AVC].Name , "AVC");

					AVC_Param_Set[i].pPrc = &Process[PROC_AVC];
					AVC_Param_Set[i].pVect = &VectorStateMach[VECT_AVC];
					AVC_Param_Set[i].VectStateNum = 1;
					AVC_Param_Set[i].Mode = 1; //BPV Mode
					AVC_Param_Set[i].MaxSpeedJog = TML_MTR_INST[TML_AX_AVC]._cfg.maxVel;

					m->pCalib->Points[CALIB_TIG_VOLT_FBK].num = 10;
					AVC_Param_Set[i].pCalibPoints		= &m->pCalib->Points[CALIB_TIG_VOLT_FBK];

				break;

			}
		}

		for(i=0 ; i < 1 ; i++){

			switch(i){

				case 0:

					strcpy(Process[m->pCfg->HeadCfg.WRST.PROC_Indx].Name , "WRST");
					strcpy(VectorStateMach[m->pCfg->HeadCfg.WRST.VECT_A_Indx].Name , "WRST");

					WRST_TML_Param_Set[i].pPrc = &Process[m->pCfg->HeadCfg.WRST.PROC_Indx];
					WRST_TML_Param_Set[i].pVect = &VectorStateMach[m->pCfg->HeadCfg.WRST.VECT_A_Indx];
					WRST_TML_Param_Set[i].VectStateNum = 1;
					WRST_TML_Param_Set[i].pTML = &TML_MTR_INST[m->pCfg->HeadCfg.WRST.TML_A_Indx] ;
					WRST_TML_Param_Set[i].Mode = 0;

					WRST_TML_Param_Set[i].GlbDirection = 1.0;

					WRST_TML_Param_Set[i].MaxAmpl = 0.0;

				break;

			}
		}

		for(i=0 ; i < 1 ; i++){

			switch(i){

				case 0:

					strcpy(Process[PROC_OSC].Name , "OSC");
					strcpy(VectorStateMach[VECT_OSC].Name , "OSC");

					OSC_TML_Param_Set[i].pPrc = &Process[PROC_OSC];
					OSC_TML_Param_Set[i].pVect = &VectorStateMach[VECT_OSC];
					OSC_TML_Param_Set[i].VectStateNum = 1;
					OSC_TML_Param_Set[i].pTML = &TML_MTR_INST[TML_AX_OSC] ;
					OSC_TML_Param_Set[i].Mode = 1; //BPV Mode

					//OSC_TML_Param_Set[i].MaxOscAmpl = 1.0 * 25.4;
					OSC_TML_Param_Set[i].MaxOscAmpl = 0.0;

				break;

			}

		}

		for(i=0 ; i < 1 ; i++){

			switch(i){

				case 0:

					strcpy(Process[PROC_GAS].Name , "GAS");
					GAS_Param_Set[i].pPrc = &Process[PROC_GAS];

					GAS_Param_Set[i].pSensInput     = &Hardware[1].Inp[5];  //FourAxis Head
					GAS_Param_Set[i].pOutput		= &Hardware[1].Outp[4];

				break;

			}

		}

		for(i=0 ; i < 1 ; i++){

			switch(i){

				case 0:

					strcpy(Process[m->pCfg->HeadCfg.INDX.PROC_Indx].Name , "INDX");
					INDEX_Param_Set[i].pPrc = &Process[m->pCfg->HeadCfg.INDX.PROC_Indx];
					//INDEX_Param_Set[i].pPrc = &Process[PROC_INDX];
					INDEX_Param_Set[i].pVect = &VectorStateMach[m->pCfg->HeadCfg.INDX.VECT_A_Indx];
					strcpy(VectorStateMach[m->pCfg->HeadCfg.INDX.VECT_A_Indx].Name , "INDX A");
					strcpy(VectorStateMach[m->pCfg->HeadCfg.INDX.VECT_B_Indx].Name , "INDX B");
					INDEX_Param_Set[i].VectStateNum = 2;
					INDEX_Param_Set[i].Mode = 0;
					INDEX_Param_Set[i].MaxSpeed = 24.0;
					INDEX_Param_Set[i].pCalibPoints		= &m->pCalib->Points[CALIB_TIG_AMPS_CMD];

				break;

			}

		}

		for(i=0 ; i < 1; i++){

			switch(i){

				case 0:

					strcpy(Process[PROC_COOL].Name , "COOLANT");
					COOL_Param_Set[i].pPrc = &Process[PROC_COOL];

					COOL_Param_Set[i].pSensInput     = &Hardware[1].Inp[4];  //FourAxis Head
					COOL_Param_Set[i].pOutput		= &Hardware[1].Outp[6];

				break;

			}

		}

		for(i=0 ; i < 1; i++){

			switch(i){

				case 0:

					strcpy(Process[PROC_HW_PS].Name , "HW PS");
					HW_PS_Param_Set[i].pPrc = &Process[PROC_HW_PS];

					HW_PS_Param_Set[i].pCalibPoints		= &m->pCalib->Points[CALIB_HW_AMPS_CMD];
					HW_PS_Param_Set[i].rawCmdMax 		= 16383.0;
					HW_PS_Param_Set[i].AmpCMD_Max 		= 160.0;

				break;

			}

		}

		for(i=0 ; i < 2; i++){

			switch(i){

				case 0:

					strcpy(Process[PROC_WIRE_FEED].Name ,"WrFeed");
					strcpy(VectorStateMach[VECT_WF].Name ,"WrFeed#1");
					strcpy(VectorStateMach[VECT_WF_1].Name ,"WrFeed#2");

					WIRE_Param_Set[i].pPrc = &Process[PROC_WIRE_FEED];
					WIRE_Param_Set[i].pVect = &VectorStateMach[VECT_WF];
					WIRE_Param_Set[i].VectStateNum = 1; //BPV Mode
					WIRE_Param_Set[i].Mode = 1;
					WIRE_Param_Set[i].MaxSpeedJog = TML_MTR_INST[TML_AX_WF]._cfg.maxVel;

					WIRE_Param_Set[i].pSynchMode = &WFSynchMode;
					WIRE_Param_Set[i].pSynchClock = &SynchClckToWF;

					WIRE_Param_Set[i].pCalibPoints	= &m->pCalib->Points[CALIB_WF_SPEED_CMD];

				break;

				case 1:

					strcpy(Process[PROC_WIRE_PULSE].Name ,"WrPulse");
					strcpy(VectorStateMach[VECT_WP].Name ,"WrPulse#1");
					strcpy(VectorStateMach[VECT_WP_1].Name ,"WrPulse#2");
					WIRE_Param_Set[i].Mode = 1; //BPV Mode

					WIRE_Param_Set[i].pPrc = &Process[PROC_WIRE_PULSE];
					WIRE_Param_Set[i].pVect = &VectorStateMach[VECT_WP];
					WIRE_Param_Set[i].VectStateNum = 1;

					WIRE_Param_Set[i].pSynchMode = &WPSynchMode;
					WIRE_Param_Set[i].pSynchClock = &SynchClckToWP;

					WIRE_Param_Set[i].pCalibPoints	= &m->pCalib->Points[CALIB_WP_SPEED_CMD];

				break;

		}

	}

		for(i=0 ; i < 1; i++){

			switch(i){

				case 0:

					strcpy(Process[PROC_TVL].Name , "TVL");
					strcpy(VectorStateMach[VECT_TVL].Name , "TVL");

					TVL_ROT_Param_Set[i].Mode = 1; //BPV Mode
					TVL_ROT_Param_Set[i].MaxSpeedJog = TML_MTR_INST[TML_AX_TVL]._cfg.maxVel;

					TVL_ROT_Param_Set[i].pPrc = &Process[PROC_TVL];
					TVL_ROT_Param_Set[i].pVect = &VectorStateMach[VECT_TVL];
					TVL_ROT_Param_Set[i].VectStateNum = 1;

					TVL_ROT_Param_Set[i].VectModeForJog = vectSt_Mode_Volt;

					TVL_ROT_Param_Set[i].TotalRescaleFactor = 1.0;
					TVL_ROT_Param_Set[i].pCalibPoints = &m->pCalib->Points[CALIB_TVL_SPEED_CMD];

					TVL_ROT_Param_Set[i].pTrackDia = &curCfg->Param[parTVL_TrackDia].val[0];
					TVL_ROT_Param_Set[i].pVelTolerance = &curCfg->Param[parTVL_SpeedTolerane].val[0];

					// TVL in Torq Mode
					TVL_ROT_Param_Set[i].VectModeForJog = vectSt_Mode_Vel;

					TVL_ROT_Param_Set[i].pEncoder = &AxisCh[TML_AX_TVL].curPos;
					TVL_ROT_Param_Set[i].pHomePos = &OLD_MTR_POS[TVL_ENC_HOME];
					TVL_ROT_Param_Set[i].EncPerTick = m->pCfg->HeadCfg.TVL.EncPerTick;
					TVL_ROT_Param_Set[i].EncDir = m->pCfg->HeadCfg.TVL.Enc_Dir;
					TVL_ROT_Param_Set[i].TicksAtHighVel = 20;

					TVL_ROT_Param_Set[i].pSynchMode = &TVLSynchMode;
					TVL_ROT_Param_Set[i].pSynchClock = &SynchClckToTVL;

			break;

	}

	}

	////////////////////////////////////////////
	/*
	Process[PROC_OSC].Disable = 1;
	Process[PROC_OSC].TestMode = 1;
	VectorStateMach[VECT_OSC].simul = 1;
	TML_MTR_INST[TML_AX_OSC].Disable = 1;
	*/

	Process[PROC_WRST].Disable = 0;
	Process[PROC_WRST].TestMode = 0;
	VectorStateMach[VECT_WRST].simul = 0;
	TML_MTR_INST[TML_AX_WRST].Disable = 0;

	////////////////////////////////////////////////////////////
	/// To jest Tylko do proby
	/*
	VectorStateMach[VECT_AVC].simul = 1;
	VectorStateMach[VECT_OSC].simul = 1;
	VectorStateMach[VECT_TVL].simul = 1;
	VectorStateMach[VECT_INDX_1].simul = 1;
	VectorStateMach[VECT_INDX_2].simul = 1;
	VectorStateMach[VECT_WF_1].simul = 1;
	VectorStateMach[VECT_WF].simul = 1;
	VectorStateMach[VECT_WP_1].simul = 1;
	VectorStateMach[VECT_WP].simul = 1;

	VectorStateMach[VECT_AVC].testMode = 1;
	VectorStateMach[VECT_OSC].testMode = 1;
	VectorStateMach[VECT_TVL].testMode = 1;
	VectorStateMach[VECT_INDX_1].testMode = 1;
	VectorStateMach[VECT_INDX_2].testMode = 1;
	VectorStateMach[VECT_WF_1].testMode = 1;
	VectorStateMach[VECT_WF].testMode = 1;
	VectorStateMach[VECT_WP_1].testMode = 1;
	VectorStateMach[VECT_WP].testMode = 1;

	TML_MTR_INST[TML_AX_AVC].Disable = 1;
	TML_MTR_INST[TML_AX_OSC].Disable = 1;
	TML_MTR_INST[TML_AX_TVL].Disable = 1;
	TML_MTR_INST[TML_AX_WRST].Disable = 1;
	TML_MTR_INST[TML_AX_WF].Disable = 1;
	TML_MTR_INST[TML_AX_WF_1].Disable = 1;
	TML_MTR_INST[TML_AX_WP].Disable = 1;
	TML_MTR_INST[TML_AX_WP_1].Disable = 1;
	////////////////////////////////////////

	Process[PROC_AVC].Disable = 1;
	Process[PROC_AVC].TestMode = 1;

	Process[PROC_INDX].Disable = 1;
	Process[PROC_INDX].TestMode = 1;

	Process[PROC_OSC].Disable = 1;
	Process[PROC_OSC].TestMode = 1;

	Process[PROC_TVL].Disable = 1;
	Process[PROC_TVL].TestMode = 1;

	Process[PROC_WIRE_FEED].Disable = 1;
	Process[PROC_WIRE_FEED].TestMode = 1;

	Process[PROC_WIRE_PULSE].Disable = 1;
	Process[PROC_WIRE_PULSE].TestMode = 1;

	Process[PROC_COOL].Disable = 1;
	Process[PROC_COOL].TestMode = 1;

	Process[PROC_GAS].Disable = 1;
	Process[PROC_GAS].TestMode = 1;
	*/

	// To tylko do proby PAMIETAC WYMAZAC
	/*
	TML_MTR_INST[TML_AX_AVC].Disable = 1;
	TML_MTR_INST[TML_AX_WF].Disable = 1;
	TML_MTR_INST[TML_AX_WP].Disable = 1;
	TML_MTR_INST[TML_AX_WRST].Disable = 1;

	Process[PROC_AVC].Disable = 1;
	*/
	////////////////////////////////////////////////////////

	return 1;

}

DINT Configure_BPV_V1_MT(MASTER_typ * m, UINT headType){
int i;

CurCfg_typ *curCfg;
Cfg_typ *cfg;
CurCalib_typ *curCalib , *defaultCalib;

	if(!m)
		return;

	curCfg = (CurCfg_typ*)m->pCurCfg;
	cfg = (Cfg_typ*)m->pCfg;

	curCalib = m->pCalib;
	defaultCalib = m->pDefaultCalib;

	if(!curCfg || !cfg || !curCalib  || !defaultCalib)
		return;

/*********************************************/
	/***   Hardware and Vectors *********************/

	TML_MTR_INST[m->pCfg->HeadCfg.TVL.TML_Indx ].pState = &VectorStateMach[m->pCfg->HeadCfg.TVL.VECT_Indx];

	TML_MTR_INST[m->pCfg->HeadCfg.AVC.TML_A_Indx ].pState = &VectorStateMach[m->pCfg->HeadCfg.AVC.VECT_A_Indx];
	TML_MTR_INST[m->pCfg->HeadCfg.AVC.TML_B_Indx ].pState = &VectorStateMach[m->pCfg->HeadCfg.AVC.VECT_B_Indx];

	TML_MTR_INST[m->pCfg->HeadCfg.OSC.TML_A_Indx ].pState = &VectorStateMach[m->pCfg->HeadCfg.OSC.VECT_A_Indx];
	TML_MTR_INST[m->pCfg->HeadCfg.OSC.TML_B_Indx ].pState = &VectorStateMach[m->pCfg->HeadCfg.OSC.VECT_B_Indx];

	TML_MTR_INST[m->pCfg->HeadCfg.WF.TML_A_Indx ].pState = &VectorStateMach[m->pCfg->HeadCfg.WF.VECT_A_Indx];
	TML_MTR_INST[m->pCfg->HeadCfg.WF.TML_B_Indx ].pState = &VectorStateMach[m->pCfg->HeadCfg.WF.VECT_B_Indx];

	TML_MTR_INST[m->pCfg->HeadCfg.WP.TML_A_Indx ].pState = &VectorStateMach[m->pCfg->HeadCfg.WP.VECT_A_Indx];
	TML_MTR_INST[m->pCfg->HeadCfg.WP.TML_B_Indx ].pState = &VectorStateMach[m->pCfg->HeadCfg.WP.VECT_B_Indx];

	TML_MTR_INST[m->pCfg->HeadCfg.WRST.TML_A_Indx ].pState = &VectorStateMach[m->pCfg->HeadCfg.WRST.VECT_A_Indx];
	TML_MTR_INST[m->pCfg->HeadCfg.WRST.TML_B_Indx ].pState = &VectorStateMach[m->pCfg->HeadCfg.WRST.VECT_B_Indx];

	DC_Mtr[m->pCfg->HeadCfg.INDX.DC_A_Indx ].pState = &VectorStateMach[m->pCfg->HeadCfg.INDX.VECT_A_Indx];
	DC_Mtr[m->pCfg->HeadCfg.INDX.DC_B_Indx ].pState = &VectorStateMach[m->pCfg->HeadCfg.INDX.VECT_B_Indx];

	/*********************************************************/
	/****   Phisical hardware configuration   ************************/

		for(i = 0 ; i < PROCESS_NUM; i++)
			strcpy(Process[i].Name , "spare");

		for(i = 0 ; i < VECTORS_NUM; i++)
			strcpy(VectorStateMach[i].Name , "spare");

			/***********************************/

		//////////////////////////////////////////////////////////////////////////////////
		// Wire Block
		for(i=0 ; i < 2; i++){

			switch(i){

				case 0:
					strcpy(Process[m->pCfg->HeadCfg.WB[i].PROC_Indx].Name , "WB_UD");
					strcpy(VectorStateMach[m->pCfg->HeadCfg.WB[i].VECT_Indx].Name , "WB_UD");

					WR_BLK_Param_Set[i].pPrc = &Process[m->pCfg->HeadCfg.WB[i].PROC_Indx];
					WR_BLK_Param_Set[i].pVect = &VectorStateMach[m->pCfg->HeadCfg.WB[i].VECT_Indx];
					WR_BLK_Param_Set[i].VectStateNum = 1;

					WR_BLK_Param_Set[i].MaxSpeedJog = 24.0;

					Gen_one = 1.0;
					WR_BLK_Param_Set[i].pJogSpeed = &Gen_one;

				break;

				case 1:
					strcpy(Process[m->pCfg->HeadCfg.WB[i].PROC_Indx].Name , "WB_LR");
					strcpy(VectorStateMach[m->pCfg->HeadCfg.WB[i].VECT_Indx].Name , "WB_LR");

					WR_BLK_Param_Set[i].pPrc = &Process[PROC_WB_LR];
					WR_BLK_Param_Set[i].pVect = &VectorStateMach[VECT_WB_LR];
					WR_BLK_Param_Set[i].VectStateNum = 1;

					WR_BLK_Param_Set[i].MaxSpeedJog = 24.0;

					Gen_one = 1.0;
					WR_BLK_Param_Set[i].pJogSpeed = &Gen_one;

				break;

			}

		}

		for(i = 0 ; i < DC2DIRMTR_NUM; i++){

			switch(i){

				case DC_WB_UD:

					strcpy(DC2DirMtr[i].Name , "WB_UD");
					DC2DirMtr[i].pState = &VectorStateMach[VECT_WB_UD];

					DC2DirMtr[i].Cfg.pQ1_output = &Hardware[1].Outp[12];
					DC2DirMtr[i].Cfg.pQ2_output = &Hardware[1].Outp[13];
					DC2DirMtr[i].Cfg.pQ3_output = &Hardware[1].Outp[14];
					DC2DirMtr[i].Cfg.pQ4_output = &Hardware[1].Outp[15];

					DC2DirMtr[i].Cfg.MtrDir = 1.0;

				break;

				case DC_WB_LR:

					strcpy(DC2DirMtr[i].Name , "WB_LR");
					DC2DirMtr[i].pState = &VectorStateMach[VECT_WB_LR];

					DC2DirMtr[i].Cfg.pQ1_output = &Hardware[1].Outp[16];
					DC2DirMtr[i].Cfg.pQ2_output = &Hardware[1].Outp[17];
					DC2DirMtr[i].Cfg.pQ3_output = &Hardware[1].Outp[18];
					DC2DirMtr[i].Cfg.pQ4_output = &Hardware[1].Outp[19];

					DC2DirMtr[i].Cfg.MtrDir = 1.0;

				break;

			}

		}
		/////////////////////////////////////////////////////////////////////////////////

		for(i = 0 ; i < GEN_MTR_NUM; i++){

			switch(i){

				case DC_INDX_1:
				case DC_INDX_2:

					switch(i){

						case DC_INDX_1:

							strcpy(DC_Mtr[i].Name , "DC INDX #1");

							DC_Mtr[i].Cfg.mtr_dir = 1.0;

							if(ProjectConfig == project_US_Orbital) // US Orbital has B and /B swapped
								DC_Mtr[i].Cfg.enc_dir = 1.0;
							else
								DC_Mtr[i].Cfg.enc_dir = -1.0;

							//DC_Mtr[i].Cfg.enc_dir = -1.0;

						break;

						case DC_INDX_2:

							strcpy(DC_Mtr[i].Name , "DC INDX #2");

							DC_Mtr[i].Cfg.mtr_dir = -1.0;

							if(ProjectConfig == project_US_Orbital) // US Orbital has B and /B swapped
								DC_Mtr[i].Cfg.enc_dir = -1.0;
							else
								DC_Mtr[i].Cfg.enc_dir = 1.0;

							//DC_Mtr[i].Cfg.enc_dir = 1.0;

						break;

					}

					//DC_Mtr[i].Cfg.units = 2000 / 59.847340050885561192713356451475; // 2000 enc ticks / 0.75 " dia * 25.4 * PI
					//DC_Mtr[i].Cfg.rev_scale = 66.0 * 0.218686666; // Ratio gear box 66:1

					DC_Mtr[i].Cfg.units =48000 / (1.25 * M_PI * 25.4); // 48000 enc ticks / 1.25 " dia * 25.4 * PI
					DC_Mtr[i].Cfg.rev_scale = 1; // Ratio gear box 66:1

					/* Parameters for PID controller */
					// To nowe
					DC_Mtr[i].msc.PIDParameters.Kp= 100.0;//0.4; //proportional gain / was 0.6
					DC_Mtr[i].msc.PIDParameters.Tn= 0.0;//0.3.1; //intergral action time
					DC_Mtr[i].msc.PIDParameters.Kfbk = 0.1; //windup dampenin

					DC_Mtr[i].msc.PID.enable = 0;
					DC_Mtr[i].msc.PID.pPar = &DC_Mtr[i].msc.PIDParameters;
					DC_Mtr[i].msc.PID.request = 3; // Read parameters from PIDParameters
					DC_Mtr[i].msc.PIDParameters.Tv= 0; //derivative action time
					DC_Mtr[i].msc.PIDParameters.Y_max = 100.0;	//max manipulated variable %
					DC_Mtr[i].msc.PIDParameters.Y_min = -100.0; //min manipulated variable %

				break;

				default:

					strcpy(DC_Mtr[i].Name , "Spare ");

				break;

			}

				//CalcUnits(&DC_Mtr[i]);
				DC_Mtr[i].msc.kPos = (float)DC_Mtr[i].Cfg.units * DC_Mtr[i].Cfg.rev_scale;

		}

		for(i = 0 ; i < TML_SERVO_NUM ; i++){

			switch(i){

				case TML_AX_TVL:

					strcpy(TML_MTR_INST[i].Name , "TVL");

					TML_MTR_INST[i]._cfg.loopPeriod = 0.001; // Slow loop
					TML_MTR_INST[i]._cfg.units = 1024 * 4; //
					TML_MTR_INST[i]._cfg.rev_motor = 73.233;
					TML_MTR_INST[i]._cfg.rev_scale = 1.0 /( 1.875 * 25.4 * M_PI) ;

					/*
					TML_MTR_INST[i]._cfg.loopPeriod = 0.0005; // Slow loop
					TML_MTR_INST[i]._cfg.units = 1024 * 4; //
					TML_MTR_INST[i]._cfg.rev_motor = 156;
					TML_MTR_INST[i]._cfg.rev_scale = 1.0 /( 1.25 * 25.4 * M_PI) ;
					*/

					TML_MTR_INST[i]._cfg.maxVel =  4500.0/60.0/TML_MTR_INST[i]._cfg.rev_motor/ TML_MTR_INST[i]._cfg.rev_scale;
					TML_MTR_INST[i]._cfg.maxAcc = TML_MTR_INST[i]._cfg.maxVel * 10.0 ;
					TML_MTR_INST[i]._cfg.absLastPos = OLD_MTR_POS[TVL_LAST_POS];
					TML_MTR_INST[i]._cfg.absFbk = 2;

					TML_MTR_INST[i]._cfg.HeartBeat = 0.08;

					/*
					strcpy(TML_MTR_INST[i]._cfg.programName , "0331_BPV_TVL.sw");
					TML_MTR_INST[i].ProgramVersion = ASC2UDINT("0331");
					*/

					strcpy(TML_MTR_INST[i]._cfg.programName , "0431_BPV_TVL_MT.sw");
					TML_MTR_INST[i].ProgramVersion = ASC2UDINT("0431");

					TML_MTR_INST[i].FirmwareVersion = ASC2UDINT("6A2B");  //0x674B
					TML_MTR_INST[i]._cfg.Appl_ID_adr = 0x7FCF;
					TML_MTR_INST[i]._cfg.NotAutoDownload = 1;

					////////////////////////////////////////////////////////

					// To jest motor z MIG Track
					/*
					strcpy(TML_MTR_INST[i].Name , "TVL");

					TML_MTR_INST[i]._cfg.loopPeriod = 0.001; // Slow loop

					// It was in BPV
					TML_MTR_INST[i]._cfg.units = 1024 * 4; //

					//TML_MTR_INST[i]._cfg.rev_motor = 156;
					//TML_MTR_INST[i]._cfg.rev_scale = 1.0 /( 1.25 * 25.4 * M_PI) ;

					TML_MTR_INST[i]._cfg.rev_motor = 73.233;
					TML_MTR_INST[i]._cfg.rev_scale = 1.0 /( 1.875 * 25.4 * M_PI) ;

					TML_MTR_INST[i]._cfg.maxVel = fabsf(4500.0/60.0/TML_MTR_INST[i]._cfg.rev_motor/ TML_MTR_INST[i]._cfg.rev_scale);
					TML_MTR_INST[i]._cfg.maxAcc = TML_MTR_INST[i]._cfg.maxVel * 10.0 ;
					//TML_MTR_INST[i]._cfg.maxAcc = TML_MTR_INST[i]._cfg.maxVel / 10.0 ;
					TML_MTR_INST[i]._cfg.absLastPos = OLD_MTR_POS[TVL_LAST_POS];
					TML_MTR_INST[i]._cfg.pAbsLastPos = &OLD_MTR_POS[TVL_LAST_POS];
					TML_MTR_INST[i]._cfg.absFbk = 3;

					TML_MTR_INST[i]._cfg.HeartBeat = 0.2;

					strcpy(TML_MTR_INST[i]._cfg.programName , "3925_BPV2_TVL_G.sw");
					TML_MTR_INST[i].ProgramVersion = ASC2UDINT("3925"); // New TVL Pos Mode with Interrupt

					TML_MTR_INST[i].FirmwareVersion = ASC2UDINT("6A2B");  //0x674B
					TML_MTR_INST[i]._cfg.Appl_ID_adr = 0x7FCF;
					TML_MTR_INST[i]._cfg.NotAutoDownload = 1;
					*/
					///////////////////////////////

				break;

				case TML_AX_OSC:

					strcpy(TML_MTR_INST[i].Name , "OSC");

					// Analog Feedback from REF
					TML_MTR_INST[i]._cfg.loopPeriod = 0.001;

					TML_MTR_INST[i]._cfg.units = 1024 * 4;
					//TML_MTR_INST[i]._cfg.rev_motor = -3.9 * 50 ;
					TML_MTR_INST[i]._cfg.rev_motor = (-75.0/19.0) * 50.0;
					TML_MTR_INST[i]._cfg.rev_scale = -1.0/ (0.625 * 25.4 *M_PI) ;

					TML_MTR_INST[i]._cfg.maxVel = 8000.0/60.0/TML_MTR_INST[i]._cfg.rev_motor/ TML_MTR_INST[i]._cfg.rev_scale;
					TML_MTR_INST[i]._cfg.maxAcc = TML_MTR_INST[i]._cfg.maxVel * 10.0 ;
					TML_MTR_INST[i]._cfg.absLastPos = OLD_MTR_POS[OSC_LAST_POS];
					TML_MTR_INST[i]._cfg.absFbk = 2;

					TML_MTR_INST[i]._cfg.HeartBeat = 0.4;
					TML_MTR_INST[i]._cfg.PVTPeriod = 0.08;

					// U_BEND_HP_PINS
					strcpy(TML_MTR_INST[i]._cfg.programName , "0322_BPV_OSC.sw");
					TML_MTR_INST[i].ProgramVersion = ASC2UDINT("0322");

					TML_MTR_INST[i].FirmwareVersion = ASC2UDINT("674C");  //0x674B
					TML_MTR_INST[i]._cfg.NotAutoDownload = 1;

					//TML_MTR_INST[i]._cfg.sftLimitPos = curCalib->Points[CALIB_OSC_SFT_LIMIT].val[0];
					//TML_MTR_INST[i]._cfg.sftLimitNeg = curCalib->Points[CALIB_OSC_SFT_LIMIT].val[1];

					//TML_MTR_INST[i]._cfg.sftLimitPos = 0.0;
					//TML_MTR_INST[i]._cfg.sftLimitNeg = 0.0;

				break;

				case TML_AX_AVC:

					strcpy(TML_MTR_INST[i].Name , "AVC");

					// Analog Feedback from REF
					TML_MTR_INST[i]._cfg.loopPeriod = 0.001;
					TML_MTR_INST[i]._cfg.units = 4096;
					TML_MTR_INST[i]._cfg.rev_motor = 1;
					TML_MTR_INST[i]._cfg.rev_scale = 1.0/5.0;
					TML_MTR_INST[i]._cfg.maxVel = 1500.0;
					TML_MTR_INST[i]._cfg.maxAcc = TML_MTR_INST[i]._cfg.maxVel * 10.0;
					//TML_MTR_INST[i]._cfg.satpMax = 27853; // KPP bylo Stauration of proportional gain
					TML_MTR_INST[i]._cfg.satpMax = 32000; // KPP bylo Stauration of proportional gain
					//TML_MTR_INST[i]._cfg.kppMax = 32000; // KPP bylo Stauration of proportional gain
					//TML_MTR_INST[i]._cfg.kipMax = 200; // KPP bylo Stauration of proportional gain
					TML_MTR_INST[i]._cfg.kppMax = 32000;
					TML_MTR_INST[i]._cfg.kipMax = 1000;
					TML_MTR_INST[i]._cfg.absFbk = 0;

					TML_MTR_INST[i]._cfg.HeartBeat = 0.8;

					TML_MTR_INST[i]._cfg.signFilter = curCfg->Param[parAVC_FbkFilter].val[0];

					//U_BEND_HP_PINS
					strcpy(TML_MTR_INST[i]._cfg.programName , "0323_BPV_AVC.sw");
					TML_MTR_INST[i].ProgramVersion = ASC2UDINT("0323");

					TML_MTR_INST[i].FirmwareVersion = ASC2UDINT("6A2B");  //0x674C , 514D
					TML_MTR_INST[i]._cfg.Appl_ID_adr = 0x7FCF;
					TML_MTR_INST[i]._cfg.NotAutoDownload = 1;

					//TML_MTR_INST[i]._cfg.sftLimitPos = 0.0;
					//TML_MTR_INST[i]._cfg.sftLimitNeg = 0.0;

					/*
					TML_MTR_INST[i]._cfg.AnalLimitPos = 3900;
					TML_MTR_INST[i]._cfg.AnalLimitNeg = 100;
					*/

					TML_MTR_INST[i]._cfg.AnalLimitPos = 0;
					TML_MTR_INST[i]._cfg.AnalLimitNeg = 0;

				break;

				case TML_AX_WRST:

					strcpy(TML_MTR_INST[i].Name , "WRIST");

					// Analog Feedback from REF
					TML_MTR_INST[i]._cfg.loopPeriod = 0.001;

					TML_MTR_INST[i]._cfg.units = 1024 * 4;
					TML_MTR_INST[i]._cfg.rev_motor = -3.9 * 50 ;
					TML_MTR_INST[i]._cfg.rev_scale = -1.0/ (0.625 * 25.4 *M_PI) ;
					TML_MTR_INST[i]._cfg.maxVel = 8000.0/60.0/TML_MTR_INST[i]._cfg.rev_motor/ TML_MTR_INST[i]._cfg.rev_scale;
					TML_MTR_INST[i]._cfg.maxAcc = TML_MTR_INST[i]._cfg.maxVel * 10.0 ;
					TML_MTR_INST[i]._cfg.absLastPos = OLD_MTR_POS[WRST_LAST_POS];
					TML_MTR_INST[i]._cfg.absFbk = 2;

					//TML_MTR_INST[i]._cfg.HeartBeat = 2.0;
					TML_MTR_INST[i]._cfg.PVTPeriod = 0.08;

					// U_BEND_HP_PINS
					//strcpy(TML_MTR_INST[i]._cfg.programName , "0334_BPV_WRST.sw");
					//TML_MTR_INST[i].ProgramVersion = ASC2UDINT("0334");

					//strcpy(TML_MTR_INST[i]._cfg.programName , "0344_BPV_WRST_OSC.sw");
					//TML_MTR_INST[i].ProgramVersion = ASC2UDINT("0344");

					strcpy(TML_MTR_INST[i]._cfg.programName , "0354_BPV_WRST_OSC_POT.sw");
					TML_MTR_INST[i].ProgramVersion = ASC2UDINT("0354");

					TML_MTR_INST[i].FirmwareVersion = ASC2UDINT("674C");  //0x674B
					//TML_MTR_INST[i]._cfg.NotAutoDownload = 1;
					TML_MTR_INST[i]._cfg.NotAutoDownload = 0;

					//TML_MTR_INST[i]._cfg.sftLimitPos = curCalib->Points[CALIB_OSC_SFT_LIMIT].val[0];
					//TML_MTR_INST[i]._cfg.sftLimitNeg = curCalib->Points[CALIB_OSC_SFT_LIMIT].val[1];

					//TML_MTR_INST[i]._cfg.sftLimitPos = 0.0;
					//TML_MTR_INST[i]._cfg.sftLimitNeg = 0.0;

				break;

				case TML_AX_WF:
				case TML_AX_WF_1:

					switch(i){

						case TML_AX_WF:

							strcpy(TML_MTR_INST[i].Name , "WF");
							TML_MTR_INST[i]._cfg.rev_scale = 1.0 /( 0.75 * 25.4 * M_PI) ;
							TML_MTR_INST[i]._cfg.rev_motor = 35.0;

						break;

						case TML_AX_WF_1:

							strcpy(TML_MTR_INST[i].Name , "WF_1");
							TML_MTR_INST[i]._cfg.rev_scale = -1.0 /( 0.75 * 25.4 * M_PI) ;
							TML_MTR_INST[i]._cfg.rev_motor = -35.0;

						break;

					}

					// Analog Feedback from REF
					TML_MTR_INST[i]._cfg.loopPeriod = 0.001;
					TML_MTR_INST[i]._cfg.units = 1024 * 4; //
					//TML_MTR_INST[i]._cfg.rev_motor = 35;

					TML_MTR_INST[i]._cfg.maxVel = 520 * 25.4/ 60.0; //// 520 ipm
					//TML_MTR_INST[i]._cfg.maxAcc = TML_MTR_INST[i]._cfg.maxVel * 100.0;
					TML_MTR_INST[i]._cfg.maxAcc = TML_MTR_INST[i]._cfg.maxVel * 4.0;
					TML_MTR_INST[i]._cfg.absFbk = 0;

					TML_MTR_INST[i]._cfg.HeartBeat = 0.4;

					strcpy(TML_MTR_INST[i]._cfg.programName , "0325_BPV_WF.sw");
					TML_MTR_INST[i].ProgramVersion = ASC2UDINT("0325");

					TML_MTR_INST[i].FirmwareVersion = ASC2UDINT("6A2B");
					TML_MTR_INST[i]._cfg.Appl_ID_adr = 0x7FCF;
					TML_MTR_INST[i]._cfg.NotAutoDownload = 1;

				break;

				case TML_AX_WP:
				case TML_AX_WP_1:

					switch(i){

						case TML_AX_WP: strcpy(TML_MTR_INST[i].Name , "WP"); break;
						case TML_AX_WP_1: strcpy(TML_MTR_INST[i].Name , "WP_1"); break;

					}

					// Analog Feedback from REF
					TML_MTR_INST[i]._cfg.loopPeriod = 0.001;

					TML_MTR_INST[i]._cfg.units = 500 * 4;
					TML_MTR_INST[i]._cfg.rev_motor = 24;
					TML_MTR_INST[i]._cfg.rev_scale = 1.0/5.0;
					TML_MTR_INST[i]._cfg.maxVel = 10000.0; //
					TML_MTR_INST[i]._cfg.maxAcc = 100.0;
					TML_MTR_INST[i]._cfg.absFbk = 0;

					TML_MTR_INST[i]._cfg.HeartBeat = 0.4;

					strcpy(TML_MTR_INST[i]._cfg.programName , "0326_BPV_WP.sw");
					TML_MTR_INST[i].ProgramVersion = ASC2UDINT("0326");

					TML_MTR_INST[i].FirmwareVersion = ASC2UDINT("6A2B");
					TML_MTR_INST[i]._cfg.Appl_ID_adr = 0x7FCF;
					TML_MTR_INST[i]._cfg.NotAutoDownload = 1;
```
